Staubli VAL3: Compensated-Y.dtx

public frame fReference = {x=1492.610, y=53.840, z=-416.740, rx=0.091, ry=-0.785, rz=-90.000, fatherId=world[0]}
public jointRx jPark = {j1=0.000, j2=0.000, j3=90.000, j4=0.000, j5=90.000, j6=0.000}
public jointRx jJoint = {j1=3.36880, j2=35.96111, j3=86.31077, j4=-179.94666, j5=-56.93914, j6=-266.65937}
public mdesc mNomSpeed = {accel=100, vel=100, decel=100, tmax=99999, rmax=99999, blend=off, leave=50, reach=50}
public mdesc mSpeed = {tmax=33.3, rmax=100, leave=0.1, reach=0.1, blend=cartesian}
public num nTraj
num nTimeStop
num nTimeStart
num nMode
num nEtat
public pointRx pPoint[1313]
  [0] = {x=-35.000, y=0.000, z=0.000, rx=-0.000, ry=0.000, rz=-0.000, shoulder=lefty, elbow=epositive, wrist=wnegative, fatherId=fReference[0]}
  [1] = {x=-34.500, y=0.000, z=-0.007, rx=-0.000, ry=0.000, rz=-0.000, shoulder=lefty, elbow=epositive, wrist=wnegative, fatherId=fReference[0]}
  [2] = {x=-34.000, y=0.000, z=-0.015, rx=-0.000, ry=0.000, rz=-0.000, shoulder=lefty, elbow=epositive, wrist=wnegative, fatherId=fReference[0]}
  [3] = {x=-33.500, y=0.000, z=-0.022, rx=-0.000, ry=0.000, rz=-0.000, shoulder=lefty, elbow=epositive, wrist=wnegative, fatherId=fReference[0]}
  [4] = {x=-32.999, y=0.000, z=-0.030, rx=-0.000, ry=0.000, rz=-0.000, shoulder=lefty, elbow=epositive, wrist=wnegative, fatherId=fReference[0]}
  [5] = {x=-32.499, y=0.000, z=-0.037, rx=-0.000, ry=0.000, rz=-0.000, shoulder=lefty, elbow=epositive, wrist=wnegative, fatherId=fReference[0]}
  [6] = {x=-31.999, y=0.000, z=-0.045, rx=-0.000, ry=0.000, rz=-0.000, shoulder=lefty, elbow=epositive, wrist=wnegative, fatherId=fReference[0]}
  [7] = {x=-31.499, y=0.000, z=-0.052, rx=-0.000, ry=0.000, rz=-0.000, shoulder=lefty, elbow=epositive, wrist=wnegative, fatherId=fReference[0]}
  [8] = {x=-30.998, y=0.000, z=-0.060, rx=-0.000, ry=0.000, rz=-0.000, shoulder=lefty, elbow=epositive, wrist=wnegative, fatherId=fReference[0]}
  [9] = {x=-30.498, y=0.000, z=-0.067, rx=-0.000, ry=0.000, rz=-0.000, shoulder=lefty, elbow=epositive, wrist=wnegative, fatherId=fReference[0]}
  [10] = {x=-29.998, y=0.000, z=-0.074, rx=-0.000, ry=0.000, rz=-0.000, shoulder=lefty, elbow=epositive, wrist=wnegative, fatherId=fReference[0]}
  [11] = {x=-29.498, y=0.000, z=-0.082, rx=-0.000, ry=0.000, rz=-0.000, shoulder=lefty, elbow=epositive, wrist=wnegative, fatherId=fReference[0]}
  [12] = {x=-28.998, y=0.000, z=-0.089, rx=-0.000, ry=0.000, rz=-0.000, shoulder=lefty, elbow=epositive, wrist=wnegative, fatherId=fReference[0]}
  [13] = {x=-28.498, y=0.000, z=-0.097, rx=-0.000, ry=0.000, rz=-0.000, shoulder=lefty, elbow=epositive, wrist=wnegative, fatherId=fReference[0]}
  [14] = {x=-27.997, y=0.000, z=-0.104, rx=-0.000, ry=0.000, rz=-0.000, shoulder=lefty, elbow=epositive, wrist=wnegative, fatherId=fReference[0]}
  [15] = {x=-27.497, y=0.000, z=-0.112, rx=-0.000, ry=0.000, rz=-0.000, shoulder=lefty, elbow=epositive, wrist=wnegative, fatherId=fReference[0]}
  [16] = {x=-26.997, y=0.000, z=-0.119, rx=-0.000, ry=0.000, rz=-0.000, shoulder=lefty, elbow=epositive, wrist=wnegative, fatherId=fReference[0]}
  [17] = {x=-26.497, y=0.000, z=-0.126, rx=-0.000, ry=0.000, rz=-0.000, shoulder=lefty, elbow=epositive, wrist=wnegative, fatherId=fReference[0]}
  [18] = {x=-25.997, y=0.000, z=-0.134, rx=-0.000, ry=0.000, rz=-0.000, shoulder=lefty, elbow=epositive, wrist=wnegative, fatherId=fReference[0]}
  [19] = {x=-25.497, y=0.000, z=-0.141, rx=-0.000, ry=0.000, rz=-0.000, shoulder=lefty, elbow=epositive, wrist=wnegative, fatherId=fReference[0]}
  [20] = {x=-24.996, y=0.000, z=-0.149, rx=-0.000, ry=0.000, rz=-0.000, shoulder=lefty, elbow=epositive, wrist=wnegative, fatherId=fReference[0]}
  [21] = {x=-24.496, y=0.000, z=-0.156, rx=-0.000, ry=0.000, rz=-0.000, shoulder=lefty, elbow=epositive, wrist=wnegative, fatherId=fReference[0]}
  [22] = {x=-23.996, y=0.000, z=-0.163, rx=-0.000, ry=0.000, rz=-0.000, shoulder=lefty, elbow=epositive, wrist=wnegative, fatherId=fReference[0]}
  [23] = {x=-23.496, y=0.000, z=-0.171, rx=-0.000, ry=0.000, rz=-0.000, shoulder=lefty, elbow=epositive, wrist=wnegative, fatherId=fReference[0]}
  [24] = {x=-22.996, y=0.000, z=-0.178, rx=-0.000, ry=0.000, rz=-0.000, shoulder=lefty, elbow=epositive, wrist=wnegative, fatherId=fReference[0]}
  [25] = {x=-22.496, y=0.000, z=-0.185, rx=-0.000, ry=0.000, rz=-0.000, shoulder=lefty, elbow=epositive, wrist=wnegative, fatherId=fReference[0]}
  [26] = {x=-21.996, y=0.000, z=-0.193, rx=-0.000, ry=0.000, rz=-0.000, shoulder=lefty, elbow=epositive, wrist=wnegative, fatherId=fReference[0]}
  [27] = {x=-21.495, y=0.000, z=-0.200, rx=-0.000, ry=0.000, rz=-0.000, shoulder=lefty, elbow=epositive, wrist=wnegative, fatherId=fReference[0]}
  [28] = {x=-20.995, y=0.000, z=-0.208, rx=-0.000, ry=0.000, rz=-0.000, shoulder=lefty, elbow=epositive, wrist=wnegative, fatherId=fReference[0]}
  [29] = {x=-20.495, y=0.000, z=-0.215, rx=-0.000, ry=0.000, rz=-0.000, shoulder=lefty, elbow=epositive, wrist=wnegative, fatherId=fReference[0]}
  [30] = {x=-19.995, y=0.000, z=-0.222, rx=-0.000, ry=0.000, rz=-0.000, shoulder=lefty, elbow=epositive, wrist=wnegative, fatherId=fReference[0]}
  [31] = {x=-19.495, y=0.000, z=-0.230, rx=-0.000, ry=0.000, rz=-0.000, shoulder=lefty, elbow=epositive, wrist=wnegative, fatherId=fReference[0]}
  [32] = {x=-18.995, y=0.000, z=-0.237, rx=-0.000, ry=0.000, rz=-0.000, shoulder=lefty, elbow=epositive, wrist=wnegative, fatherId=fReference[0]}
  [33] = {x=-18.495, y=0.000, z=-0.244, rx=-0.000, ry=0.000, rz=-0.000, shoulder=lefty, elbow=epositive, wrist=wnegative, fatherId=fReference[0]}
  [34] = {x=-17.995, y=0.000, z=-0.252, rx=-0.000, ry=0.000, rz=-0.000, shoulder=lefty, elbow=epositive, wrist=wnegative, fatherId=fReference[0]}
  [35] = {x=-17.494, y=0.000, z=-0.259, rx=-0.000, ry=0.000, rz=-0.000, shoulder=lefty, elbow=epositive, wrist=wnegative, fatherId=fReference[0]}
  [36] = {x=-16.994, y=0.000, z=-0.266, rx=-0.000, ry=0.000, rz=-0.000, shoulder=lefty, elbow=epositive, wrist=wnegative, fatherId=fReference[0]}
  [37] = {x=-16.494, y=0.000, z=-0.274, rx=-0.000, ry=0.000, rz=-0.000, shoulder=lefty, elbow=epositive, wrist=wnegative, fatherId=fReference[0]}
  [38] = {x=-15.994, y=0.000, z=-0.281, rx=-0.000, ry=0.000, rz=-0.000, shoulder=lefty, elbow=epositive, wrist=wnegative, fatherId=fReference[0]}
  [39] = {x=-15.494, y=0.000, z=-0.288, rx=-0.000, ry=0.000, rz=-0.000, shoulder=lefty, elbow=epositive, wrist=wnegative, fatherId=fReference[0]}
  [40] = {x=-14.994, y=0.000, z=-0.296, rx=-0.000, ry=0.000, rz=-0.000, shoulder=lefty, elbow=epositive, wrist=wnegative, fatherId=fReference[0]}
  [41] = {x=-14.494, y=0.000, z=-0.303, rx=-0.000, ry=0.000, rz=-0.000, shoulder=lefty, elbow=epositive, wrist=wnegative, fatherId=fReference[0]}
  [42] = {x=-13.994, y=0.000, z=-0.310, rx=-0.000, ry=0.000, rz=-0.000, shoulder=lefty, elbow=epositive, wrist=wnegative, fatherId=fReference[0]}
  [43] = {x=-13.493, y=0.000, z=-0.318, rx=-0.000, ry=0.000, rz=-0.000, shoulder=lefty, elbow=epositive, wrist=wnegative, fatherId=fReference[0]}
  [44] = {x=-12.993, y=0.000, z=-0.325, rx=-0.000, ry=0.000, rz=-0.000, shoulder=lefty, elbow=epositive, wrist=wnegative, fatherId=fReference[0]}
  [45] = {x=-12.493, y=0.000, z=-0.332, rx=-0.000, ry=0.000, rz=-0.000, shoulder=lefty, elbow=epositive, wrist=wnegative, fatherId=fReference[0]}
  [46] = {x=-11.993, y=0.000, z=-0.340, rx=-0.000, ry=0.000, rz=-0.000, shoulder=lefty, elbow=epositive, wrist=wnegative, fatherId=fReference[0]}
  [47] = {x=-11.493, y=0.000, z=-0.347, rx=-0.000, ry=0.000, rz=-0.000, shoulder=lefty, elbow=epositive, wrist=wnegative, fatherId=fReference[0]}
  [48] = {x=-10.993, y=0.000, z=-0.354, rx=-0.000, ry=0.000, rz=-0.000, shoulder=lefty, elbow=epositive, wrist=wnegative, fatherId=fReference[0]}
  [49] = {x=-10.493, y=0.000, z=-0.362, rx=-0.000, ry=0.000, rz=-0.000, shoulder=lefty, elbow=epositive, wrist=wnegative, fatherId=fReference[0]}
  [50] = {x=-9.993, y=0.000, z=-0.369, rx=-0.000, ry=0.000, rz=-0.000, shoulder=lefty, elbow=epositive, wrist=wnegative, fatherId=fReference[0]}
  [51] = {x=-9.492, y=0.000, z=-0.377, rx=-0.000, ry=0.000, rz=-0.000, shoulder=lefty, elbow=epositive, wrist=wnegative, fatherId=fReference[0]}
  [52] = {x=-8.992, y=0.000, z=-0.384, rx=-0.000, ry=0.000, rz=-0.000, shoulder=lefty, elbow=epositive, wrist=wnegative, fatherId=fReference[0]}
  [53] = {x=-8.492, y=0.000, z=-0.391, rx=-0.000, ry=0.000, rz=-0.000, shoulder=lefty, elbow=epositive, wrist=wnegative, fatherId=fReference[0]}
  [54] = {x=-7.992, y=0.000, z=-0.399, rx=-0.000, ry=0.000, rz=-0.000, shoulder=lefty, elbow=epositive, wrist=wnegative, fatherId=fReference[0]}
  [55] = {x=-7.492, y=0.000, z=-0.406, rx=-0.000, ry=0.000, rz=-0.000, shoulder=lefty, elbow=epositive, wrist=wnegative, fatherId=fReference[0]}
  [56] = {x=-6.992, y=0.000, z=-0.413, rx=-0.000, ry=0.000, rz=-0.000, shoulder=lefty, elbow=epositive, wrist=wnegative, fatherId=fReference[0]}
  [57] = {x=-6.492, y=0.000, z=-0.421, rx=-0.000, ry=0.000, rz=-0.000, shoulder=lefty, elbow=epositive, wrist=wnegative, fatherId=fReference[0]}
  [58] = {x=-5.991, y=0.000, z=-0.428, rx=-0.000, ry=0.000, rz=-0.000, shoulder=lefty, elbow=epositive, wrist=wnegative, fatherId=fReference[0]}
  [59] = {x=-5.491, y=0.000, z=-0.435, rx=-0.000, ry=0.000, rz=-0.000, shoulder=lefty, elbow=epositive, wrist=wnegative, fatherId=fReference[0]}
  [60] = {x=-4.991, y=0.000, z=-0.443, rx=-0.000, ry=0.000, rz=-0.000, shoulder=lefty, elbow=epositive, wrist=wnegative, fatherId=fReference[0]}
  [61] = {x=-4.491, y=0.000, z=-0.450, rx=-0.000, ry=0.000, rz=-0.000, shoulder=lefty, elbow=epositive, wrist=wnegative, fatherId=fReference[0]}
  [62] = {x=-3.991, y=0.000, z=-0.458, rx=-0.000, ry=0.000, rz=-0.000, shoulder=lefty, elbow=epositive, wrist=wnegative, fatherId=fReference[0]}
  [63] = {x=-3.491, y=0.000, z=-0.465, rx=-0.000, ry=0.000, rz=-0.000, shoulder=lefty, elbow=epositive, wrist=wnegative, fatherId=fReference[0]}
  [64] = {x=-2.991, y=0.000, z=-0.472, rx=-0.000, ry=0.000, rz=-0.000, shoulder=lefty, elbow=epositive, wrist=wnegative, fatherId=fReference[0]}
  [65] = {x=-2.490, y=0.000, z=-0.480, rx=-0.000, ry=0.000, rz=-0.000, shoulder=lefty, elbow=epositive, wrist=wnegative, fatherId=fReference[0]}
  [66] = {x=-1.990, y=0.000, z=-0.487, rx=-0.000, ry=0.000, rz=-0.000, shoulder=lefty, elbow=epositive, wrist=wnegative, fatherId=fReference[0]}
  [67] = {x=-1.490, y=0.000, z=-0.495, rx=-0.000, ry=0.000, rz=-0.000, shoulder=lefty, elbow=epositive, wrist=wnegative, fatherId=fReference[0]}
  [68] = {x=-0.990, y=0.000, z=-0.502, rx=-0.000, ry=0.000, rz=-0.000, shoulder=lefty, elbow=epositive, wrist=wnegative, fatherId=fReference[0]}
  [69] = {x=-0.490, y=0.000, z=-0.509, rx=-0.000, ry=0.000, rz=-0.000, shoulder=lefty, elbow=epositive, wrist=wnegative, fatherId=fReference[0]}
  [70] = {x=0.010, y=0.000, z=-0.517, rx=-0.000, ry=0.000, rz=-0.000, shoulder=lefty, elbow=epositive, wrist=wnegative, fatherId=fReference[0]}
  [71] = {x=0.511, y=0.000, z=-0.524, rx=-0.000, ry=0.000, rz=-0.000, shoulder=lefty, elbow=epositive, wrist=wnegative, fatherId=fReference[0]}
  [72] = {x=1.011, y=0.000, z=-0.532, rx=-0.000, ry=0.000, rz=-0.000, shoulder=lefty, elbow=epositive, wrist=wnegative, fatherId=fReference[0]}
  [73] = {x=1.511, y=0.000, z=-0.539, rx=-0.000, ry=0.000, rz=-0.000, shoulder=lefty, elbow=epositive, wrist=wnegative, fatherId=fReference[0]}
  [74] = {x=2.011, y=0.000, z=-0.547, rx=-0.000, ry=0.000, rz=-0.000, shoulder=lefty, elbow=epositive, wrist=wnegative, fatherId=fReference[0]}
  [75] = {x=2.511, y=0.000, z=-0.554, rx=-0.000, ry=0.000, rz=-0.000, shoulder=lefty, elbow=epositive, wrist=wnegative, fatherId=fReference[0]}
  [76] = {x=3.012, y=0.000, z=-0.562, rx=-0.000, ry=0.000, rz=-0.000, shoulder=lefty, elbow=epositive, wrist=wnegative, fatherId=fReference[0]}
  [77] = {x=3.512, y=0.000, z=-0.569, rx=-0.000, ry=0.000, rz=-0.000, shoulder=lefty, elbow=epositive, wrist=wnegative, fatherId=fReference[0]}
  [78] = {x=4.012, y=0.000, z=-0.576, rx=-0.000, ry=0.000, rz=-0.000, shoulder=lefty, elbow=epositive, wrist=wnegative, fatherId=fReference[0]}
  [79] = {x=4.512, y=0.000, z=-0.584, rx=-0.000, ry=0.000, rz=-0.000, shoulder=lefty, elbow=epositive, wrist=wnegative, fatherId=fReference[0]}
  [80] = {x=5.012, y=0.000, z=-0.591, rx=-0.000, ry=0.000, rz=-0.000, shoulder=lefty, elbow=epositive, wrist=wnegative, fatherId=fReference[0]}
  [81] = {x=5.513, y=0.000, z=-0.599, rx=-0.000, ry=0.000, rz=-0.000, shoulder=lefty, elbow=epositive, wrist=wnegative, fatherId=fReference[0]}
  [82] = {x=6.013, y=0.000, z=-0.606, rx=-0.000, ry=0.000, rz=-0.000, shoulder=lefty, elbow=epositive, wrist=wnegative, fatherId=fReference[0]}
  [83] = {x=6.513, y=0.000, z=-0.614, rx=-0.000, ry=0.000, rz=-0.000, shoulder=lefty, elbow=epositive, wrist=wnegative, fatherId=fReference[0]}
  [84] = {x=7.013, y=0.000, z=-0.621, rx=-0.000, ry=0.000, rz=-0.000, shoulder=lefty, elbow=epositive, wrist=wnegative, fatherId=fReference[0]}
  [85] = {x=7.514, y=0.000, z=-0.629, rx=-0.000, ry=0.000, rz=-0.000, shoulder=lefty, elbow=epositive, wrist=wnegative, fatherId=fReference[0]}
  [86] = {x=8.014, y=0.000, z=-0.637, rx=-0.000, ry=0.000, rz=-0.000, shoulder=lefty, elbow=epositive, wrist=wnegative, fatherId=fReference[0]}
  [87] = {x=8.514, y=0.000, z=-0.644, rx=-0.000, ry=0.000, rz=-0.000, shoulder=lefty, elbow=epositive, wrist=wnegative, fatherId=fReference[0]}
  [88] = {x=9.014, y=0.000, z=-0.652, rx=-0.000, ry=0.000, rz=-0.000, shoulder=lefty, elbow=epositive, wrist=wnegative, fatherId=fReference[0]}
  [89] = {x=9.515, y=0.000, z=-0.659, rx=-0.000, ry=0.000, rz=-0.000, shoulder=lefty, elbow=epositive, wrist=wnegative, fatherId=fReference[0]}
  [90] = {x=10.015, y=0.000, z=-0.667, rx=-0.000, ry=0.000, rz=-0.000, shoulder=lefty, elbow=epositive, wrist=wnegative, fatherId=fReference[0]}
  [91] = {x=10.515, y=0.000, z=-0.674, rx=-0.000, ry=0.000, rz=-0.000, shoulder=lefty, elbow=epositive, wrist=wnegative, fatherId=fReference[0]}
  [92] = {x=11.016, y=0.000, z=-0.682, rx=-0.000, ry=0.000, rz=-0.000, shoulder=lefty, elbow=epositive, wrist=wnegative, fatherId=fReference[0]}
  [93] = {x=11.516, y=0.000, z=-0.690, rx=-0.000, ry=0.000, rz=-0.000, shoulder=lefty, elbow=epositive, wrist=wnegative, fatherId=fReference[0]}
  [94] = {x=12.016, y=0.000, z=-0.697, rx=-0.000, ry=0.000, rz=-0.000, shoulder=lefty, elbow=epositive, wrist=wnegative, fatherId=fReference[0]}
  [95] = {x=12.516, y=0.000, z=-0.705, rx=-0.000, ry=0.000, rz=-0.000, shoulder=lefty, elbow=epositive, wrist=wnegative, fatherId=fReference[0]}
  [96] = {x=13.017, y=0.000, z=-0.713, rx=-0.000, ry=0.000, rz=-0.000, shoulder=lefty, elbow=epositive, wrist=wnegative, fatherId=fReference[0]}
  [97] = {x=13.517, y=0.000, z=-0.720, rx=-0.000, ry=0.000, rz=-0.000, shoulder=lefty, elbow=epositive, wrist=wnegative, fatherId=fReference[0]}
  [98] = {x=14.017, y=0.000, z=-0.728, rx=-0.000, ry=0.000, rz=-0.000, shoulder=lefty, elbow=epositive, wrist=wnegative, fatherId=fReference[0]}
  [99] = {x=14.518, y=0.000, z=-0.736, rx=-0.000, ry=0.000, rz=-0.000, shoulder=lefty, elbow=epositive, wrist=wnegative, fatherId=fReference[0]}
  [100] = {x=15.018, y=0.000, z=-0.743, rx=-0.000, ry=0.000, rz=-0.000, shoulder=lefty, elbow=epositive, wrist=wnegative, fatherId=fReference[0]}
  [101] = {x=15.519, y=0.000, z=-0.751, rx=-0.000, ry=0.000, rz=-0.000, shoulder=lefty, elbow=epositive, wrist=wnegative, fatherId=fReference[0]}
  [102] = {x=16.019, y=0.000, z=-0.759, rx=-0.000, ry=0.000, rz=-0.000, shoulder=lefty, elbow=epositive, wrist=wnegative, fatherId=fReference[0]}
  [103] = {x=16.519, y=0.000, z=-0.766, rx=-0.000, ry=0.000, rz=-0.000, shoulder=lefty, elbow=epositive, wrist=wnegative, fatherId=fReference[0]}
  [104] = {x=17.020, y=0.000, z=-0.774, rx=-0.000, ry=0.000, rz=-0.000, shoulder=lefty, elbow=epositive, wrist=wnegative, fatherId=fReference[0]}
  [105] = {x=17.520, y=0.000, z=-0.782, rx=-0.000, ry=0.000, rz=-0.000, shoulder=lefty, elbow=epositive, wrist=wnegative, fatherId=fReference[0]}
  [106] = {x=18.020, y=0.000, z=-0.790, rx=-0.000, ry=0.000, rz=-0.000, shoulder=lefty, elbow=epositive, wrist=wnegative, fatherId=fReference[0]}
  [107] = {x=18.521, y=0.000, z=-0.798, rx=-0.000, ry=0.000, rz=-0.000, shoulder=lefty, elbow=epositive, wrist=wnegative, fatherId=fReference[0]}
  [108] = {x=19.021, y=0.000, z=-0.805, rx=-0.000, ry=0.000, rz=-0.000, shoulder=lefty, elbow=epositive, wrist=wnegative, fatherId=fReference[0]}
  [109] = {x=19.522, y=0.000, z=-0.813, rx=-0.000, ry=0.000, rz=-0.000, shoulder=lefty, elbow=epositive, wrist=wnegative, fatherId=fReference[0]}
  [110] = {x=20.022, y=0.000, z=-0.821, rx=-0.000, ry=0.000, rz=-0.000, shoulder=lefty, elbow=epositive, wrist=wnegative, fatherId=fReference[0]}
  [111] = {x=20.523, y=0.000, z=-0.829, rx=-0.000, ry=0.000, rz=-0.000, shoulder=lefty, elbow=epositive, wrist=wnegative, fatherId=fReference[0]}
  [112] = {x=21.023, y=0.000, z=-0.837, rx=-0.000, ry=0.000, rz=-0.000, shoulder=lefty, elbow=epositive, wrist=wnegative, fatherId=fReference[0]}
  [113] = {x=21.524, y=0.000, z=-0.845, rx=-0.000, ry=0.000, rz=-0.000, shoulder=lefty, elbow=epositive, wrist=wnegative, fatherId=fReference[0]}
  [114] = {x=22.024, y=0.000, z=-0.853, rx=-0.000, ry=0.000, rz=-0.000, shoulder=lefty, elbow=epositive, wrist=wnegative, fatherId=fReference[0]}
  [115] = {x=22.525, y=0.000, z=-0.861, rx=-0.000, ry=0.000, rz=-0.000, shoulder=lefty, elbow=epositive, wrist=wnegative, fatherId=fReference[0]}
  [116] = {x=23.025, y=0.000, z=-0.869, rx=-0.000, ry=0.000, rz=-0.000, shoulder=lefty, elbow=epositive, wrist=wnegative, fatherId=fReference[0]}
  [117] = {x=23.526, y=0.000, z=-0.877, rx=-0.000, ry=0.000, rz=-0.000, shoulder=lefty, elbow=epositive, wrist=wnegative, fatherId=fReference[0]}
  [118] = {x=24.026, y=0.000, z=-0.885, rx=-0.000, ry=0.000, rz=-0.000, shoulder=lefty, elbow=epositive, wrist=wnegative, fatherId=fReference[0]}
  [119] = {x=24.527, y=0.000, z=-0.893, rx=-0.000, ry=0.000, rz=-0.000, shoulder=lefty, elbow=epositive, wrist=wnegative, fatherId=fReference[0]}
  [120] = {x=25.028, y=0.000, z=-0.901, rx=-0.000, ry=0.000, rz=-0.000, shoulder=lefty, elbow=epositive, wrist=wnegative, fatherId=fReference[0]}
  [121] = {x=25.528, y=0.000, z=-0.909, rx=-0.000, ry=0.000, rz=-0.000, shoulder=lefty, elbow=epositive, wrist=wnegative, fatherId=fReference[0]}
  [122] = {x=26.029, y=0.000, z=-0.917, rx=-0.000, ry=0.000, rz=-0.000, shoulder=lefty, elbow=epositive, wrist=wnegative, fatherId=fReference[0]}
  [123] = {x=26.530, y=0.000, z=-0.925, rx=-0.000, ry=0.000, rz=-0.000, shoulder=lefty, elbow=epositive, wrist=wnegative, fatherId=fReference[0]}
  [124] = {x=27.030, y=0.000, z=-0.933, rx=-0.000, ry=0.000, rz=-0.000, shoulder=lefty, elbow=epositive, wrist=wnegative, fatherId=fReference[0]}
  [125] = {x=27.531, y=0.000, z=-0.941, rx=-0.000, ry=0.000, rz=-0.000, shoulder=lefty, elbow=epositive, wrist=wnegative, fatherId=fReference[0]}
  [126] = {x=28.032, y=0.000, z=-0.950, rx=-0.000, ry=0.000, rz=-0.000, shoulder=lefty, elbow=epositive, wrist=wnegative, fatherId=fReference[0]}
  [127] = {x=28.532, y=0.000, z=-0.958, rx=-0.000, ry=0.000, rz=-0.000, shoulder=lefty, elbow=epositive, wrist=wnegative, fatherId=fReference[0]}
  [128] = {x=29.033, y=0.000, z=-0.966, rx=-0.000, ry=0.000, rz=-0.000, shoulder=lefty, elbow=epositive, wrist=wnegative, fatherId=fReference[0]}
  [129] = {x=29.534, y=0.000, z=-0.974, rx=-0.000, ry=0.000, rz=-0.000, shoulder=lefty, elbow=epositive, wrist=wnegative, fatherId=fReference[0]}
  [130] = {x=30.035, y=0.000, z=-0.983, rx=-0.000, ry=0.000, rz=-0.000, shoulder=lefty, elbow=epositive, wrist=wnegative, fatherId=fReference[0]}
  [131] = {x=30.536, y=0.000, z=-0.991, rx=-0.000, ry=0.000, rz=-0.000, shoulder=lefty, elbow=epositive, wrist=wnegative, fatherId=fReference[0]}
  [132] = {x=31.036, y=0.000, z=-1.000, rx=-0.000, ry=0.000, rz=-0.000, shoulder=lefty, elbow=epositive, wrist=wnegative, fatherId=fReference[0]}
  [133] = {x=31.537, y=0.000, z=-1.008, rx=-0.000, ry=0.000, rz=-0.000, shoulder=lefty, elbow=epositive, wrist=wnegative, fatherId=fReference[0]}
  [134] = {x=32.038, y=0.000, z=-1.016, rx=-0.000, ry=0.000, rz=-0.000, shoulder=lefty, elbow=epositive, wrist=wnegative, fatherId=fReference[0]}
  [135] = {x=32.539, y=0.000, z=-1.025, rx=-0.000, ry=0.000, rz=-0.000, shoulder=lefty, elbow=epositive, wrist=wnegative, fatherId=fReference[0]}
  [136] = {x=33.040, y=0.000, z=-1.034, rx=-0.000, ry=0.000, rz=-0.000, shoulder=lefty, elbow=epositive, wrist=wnegative, fatherId=fReference[0]}
  [137] = {x=33.541, y=0.000, z=-1.042, rx=-0.000, ry=0.000, rz=-0.000, shoulder=lefty, elbow=epositive, wrist=wnegative, fatherId=fReference[0]}
  [138] = {x=34.042, y=0.000, z=-1.051, rx=-0.000, ry=0.000, rz=-0.000, shoulder=lefty, elbow=epositive, wrist=wnegative, fatherId=fReference[0]}
  [139] = {x=34.543, y=0.000, z=-1.060, rx=-0.000, ry=0.000, rz=-0.000, shoulder=lefty, elbow=epositive, wrist=wnegative, fatherId=fReference[0]}
  [140] = {x=35.026, y=0.000, z=-1.067, rx=-0.000, ry=0.000, rz=-0.000, shoulder=lefty, elbow=epositive, wrist=wnegative, fatherId=fReference[0]}
  [141] = {x=34.526, y=0.000, z=-1.073, rx=-0.000, ry=0.000, rz=-0.000, shoulder=lefty, elbow=epositive, wrist=wnegative, fatherId=fReference[0]}
  [142] = {x=34.026, y=0.000, z=-1.080, rx=-0.000, ry=0.000, rz=-0.000, shoulder=lefty, elbow=epositive, wrist=wnegative, fatherId=fReference[0]}
  [143] = {x=33.525, y=0.000, z=-1.086, rx=-0.000, ry=0.000, rz=-0.000, shoulder=lefty, elbow=epositive, wrist=wnegative, fatherId=fReference[0]}
  [144] = {x=33.025, y=0.000, z=-1.093, rx=-0.000, ry=0.000, rz=-0.000, shoulder=lefty, elbow=epositive, wrist=wnegative, fatherId=fReference[0]}
  [145] = {x=32.525, y=0.000, z=-1.100, rx=-0.000, ry=0.000, rz=-0.000, shoulder=lefty, elbow=epositive, wrist=wnegative, fatherId=fReference[0]}
  [146] = {x=32.025, y=0.000, z=-1.107, rx=-0.000, ry=0.000, rz=-0.000, shoulder=lefty, elbow=epositive, wrist=wnegative, fatherId=fReference[0]}
  [147] = {x=31.524, y=0.000, z=-1.114, rx=-0.000, ry=0.000, rz=-0.000, shoulder=lefty, elbow=epositive, wrist=wnegative, fatherId=fReference[0]}
  [148] = {x=31.024, y=0.000, z=-1.121, rx=-0.000, ry=0.000, rz=-0.000, shoulder=lefty, elbow=epositive, wrist=wnegative, fatherId=fReference[0]}
  [149] = {x=30.524, y=0.000, z=-1.127, rx=-0.000, ry=0.000, rz=-0.000, shoulder=lefty, elbow=epositive, wrist=wnegative, fatherId=fReference[0]}
  [150] = {x=30.024, y=0.000, z=-1.135, rx=-0.000, ry=0.000, rz=-0.000, shoulder=lefty, elbow=epositive, wrist=wnegative, fatherId=fReference[0]}
  [151] = {x=29.524, y=0.000, z=-1.141, rx=-0.000, ry=0.000, rz=-0.000, shoulder=lefty, elbow=epositive, wrist=wnegative, fatherId=fReference[0]}
  [152] = {x=29.024, y=0.000, z=-1.149, rx=-0.000, ry=0.000, rz=-0.000, shoulder=lefty, elbow=epositive, wrist=wnegative, fatherId=fReference[0]}
  [153] = {x=28.523, y=0.000, z=-1.155, rx=-0.000, ry=0.000, rz=-0.000, shoulder=lefty, elbow=epositive, wrist=wnegative, fatherId=fReference[0]}
  [154] = {x=28.023, y=0.000, z=-1.163, rx=-0.000, ry=0.000, rz=-0.000, shoulder=lefty, elbow=epositive, wrist=wnegative, fatherId=fReference[0]}
  [155] = {x=27.523, y=0.000, z=-1.170, rx=-0.000, ry=0.000, rz=-0.000, shoulder=lefty, elbow=epositive, wrist=wnegative, fatherId=fReference[0]}
  [156] = {x=27.023, y=0.000, z=-1.177, rx=-0.000, ry=0.000, rz=-0.000, shoulder=lefty, elbow=epositive, wrist=wnegative, fatherId=fReference[0]}
  [157] = {x=26.523, y=0.000, z=-1.184, rx=-0.000, ry=0.000, rz=-0.000, shoulder=lefty, elbow=epositive, wrist=wnegative, fatherId=fReference[0]}
  [158] = {x=26.023, y=0.000, z=-1.191, rx=-0.000, ry=0.000, rz=-0.000, shoulder=lefty, elbow=epositive, wrist=wnegative, fatherId=fReference[0]}
  [159] = {x=25.523, y=0.000, z=-1.198, rx=-0.000, ry=0.000, rz=-0.000, shoulder=lefty, elbow=epositive, wrist=wnegative, fatherId=fReference[0]}
  [160] = {x=25.023, y=0.000, z=-1.205, rx=-0.000, ry=0.000, rz=-0.000, shoulder=lefty, elbow=epositive, wrist=wnegative, fatherId=fReference[0]}
  [161] = {x=24.523, y=0.000, z=-1.212, rx=-0.000, ry=0.000, rz=-0.000, shoulder=lefty, elbow=epositive, wrist=wnegative, fatherId=fReference[0]}
  [162] = {x=24.023, y=0.000, z=-1.219, rx=-0.000, ry=0.000, rz=-0.000, shoulder=lefty, elbow=epositive, wrist=wnegative, fatherId=fReference[0]}
  [163] = {x=23.523, y=0.000, z=-1.227, rx=-0.000, ry=0.000, rz=-0.000, shoulder=lefty, elbow=epositive, wrist=wnegative, fatherId=fReference[0]}
  [164] = {x=23.023, y=0.000, z=-1.234, rx=-0.000, ry=0.000, rz=-0.000, shoulder=lefty, elbow=epositive, wrist=wnegative, fatherId=fReference[0]}
  [165] = {x=22.523, y=0.000, z=-1.241, rx=-0.000, ry=0.000, rz=-0.000, shoulder=lefty, elbow=epositive, wrist=wnegative, fatherId=fReference[0]}
  [166] = {x=22.022, y=0.000, z=-1.248, rx=-0.000, ry=0.000, rz=-0.000, shoulder=lefty, elbow=epositive, wrist=wnegative, fatherId=fReference[0]}
  [167] = {x=21.522, y=0.000, z=-1.255, rx=-0.000, ry=0.000, rz=-0.000, shoulder=lefty, elbow=epositive, wrist=wnegative, fatherId=fReference[0]}
  [168] = {x=21.022, y=0.000, z=-1.262, rx=-0.000, ry=0.000, rz=-0.000, shoulder=lefty, elbow=epositive, wrist=wnegative, fatherId=fReference[0]}
  [169] = {x=20.522, y=0.000, z=-1.270, rx=-0.000, ry=0.000, rz=-0.000, shoulder=lefty, elbow=epositive, wrist=wnegative, fatherId=fReference[0]}
  [170] = {x=20.022, y=0.000, z=-1.277, rx=-0.000, ry=0.000, rz=-0.000, shoulder=lefty, elbow=epositive, wrist=wnegative, fatherId=fReference[0]}
  [171] = {x=19.522, y=0.000, z=-1.284, rx=-0.000, ry=0.000, rz=-0.000, shoulder=lefty, elbow=epositive, wrist=wnegative, fatherId=fReference[0]}
  [172] = {x=19.022, y=0.000, z=-1.292, rx=-0.000, ry=0.000, rz=-0.000, shoulder=lefty, elbow=epositive, wrist=wnegative, fatherId=fReference[0]}
  [173] = {x=18.522, y=0.000, z=-1.299, rx=-0.000, ry=0.000, rz=-0.000, shoulder=lefty, elbow=epositive, wrist=wnegative, fatherId=fReference[0]}
  [174] = {x=18.022, y=0.000, z=-1.306, rx=-0.000, ry=0.000, rz=-0.000, shoulder=lefty, elbow=epositive, wrist=wnegative, fatherId=fReference[0]}
  [175] = {x=17.522, y=0.000, z=-1.313, rx=-0.000, ry=0.000, rz=-0.000, shoulder=lefty, elbow=epositive, wrist=wnegative, fatherId=fReference[0]}
  [176] = {x=17.022, y=0.000, z=-1.321, rx=-0.000, ry=0.000, rz=-0.000, shoulder=lefty, elbow=epositive, wrist=wnegative, fatherId=fReference[0]}
  [177] = {x=16.522, y=0.000, z=-1.328, rx=-0.000, ry=0.000, rz=-0.000, shoulder=lefty, elbow=epositive, wrist=wnegative, fatherId=fReference[0]}
  [178] = {x=16.022, y=0.000, z=-1.335, rx=-0.000, ry=0.000, rz=-0.000, shoulder=lefty, elbow=epositive, wrist=wnegative, fatherId=fReference[0]}
  [179] = {x=15.522, y=0.000, z=-1.343, rx=-0.000, ry=0.000, rz=-0.000, shoulder=lefty, elbow=epositive, wrist=wnegative, fatherId=fReference[0]}
  [180] = {x=15.022, y=0.000, z=-1.350, rx=-0.000, ry=0.000, rz=-0.000, shoulder=lefty, elbow=epositive, wrist=wnegative, fatherId=fReference[0]}
  [181] = {x=14.522, y=0.000, z=-1.357, rx=-0.000, ry=0.000, rz=-0.000, shoulder=lefty, elbow=epositive, wrist=wnegative, fatherId=fReference[0]}
  [182] = {x=14.022, y=0.000, z=-1.365, rx=-0.000, ry=0.000, rz=-0.000, shoulder=lefty, elbow=epositive, wrist=wnegative, fatherId=fReference[0]}
  [183] = {x=13.523, y=0.000, z=-1.372, rx=-0.000, ry=0.000, rz=-0.000, shoulder=lefty, elbow=epositive, wrist=wnegative, fatherId=fReference[0]}
  [184] = {x=13.023, y=0.000, z=-1.380, rx=-0.000, ry=0.000, rz=-0.000, shoulder=lefty, elbow=epositive, wrist=wnegative, fatherId=fReference[0]}
  [185] = {x=12.523, y=0.000, z=-1.387, rx=-0.000, ry=0.000, rz=-0.000, shoulder=lefty, elbow=epositive, wrist=wnegative, fatherId=fReference[0]}
  [186] = {x=12.023, y=0.000, z=-1.395, rx=-0.000, ry=0.000, rz=-0.000, shoulder=lefty, elbow=epositive, wrist=wnegative, fatherId=fReference[0]}
  [187] = {x=11.523, y=0.000, z=-1.402, rx=-0.000, ry=0.000, rz=-0.000, shoulder=lefty, elbow=epositive, wrist=wnegative, fatherId=fReference[0]}
  [188] = {x=11.023, y=0.000, z=-1.409, rx=-0.000, ry=0.000, rz=-0.000, shoulder=lefty, elbow=epositive, wrist=wnegative, fatherId=fReference[0]}
  [189] = {x=10.523, y=0.000, z=-1.417, rx=-0.000, ry=0.000, rz=-0.000, shoulder=lefty, elbow=epositive, wrist=wnegative, fatherId=fReference[0]}
  [190] = {x=10.023, y=0.000, z=-1.424, rx=-0.000, ry=0.000, rz=-0.000, shoulder=lefty, elbow=epositive, wrist=wnegative, fatherId=fReference[0]}
  [191] = {x=9.523, y=0.000, z=-1.432, rx=-0.000, ry=0.000, rz=-0.000, shoulder=lefty, elbow=epositive, wrist=wnegative, fatherId=fReference[0]}
  [192] = {x=9.023, y=0.000, z=-1.439, rx=-0.000, ry=0.000, rz=-0.000, shoulder=lefty, elbow=epositive, wrist=wnegative, fatherId=fReference[0]}
  [193] = {x=8.523, y=0.000, z=-1.447, rx=-0.000, ry=0.000, rz=-0.000, shoulder=lefty, elbow=epositive, wrist=wnegative, fatherId=fReference[0]}
  [194] = {x=8.023, y=0.000, z=-1.454, rx=-0.000, ry=0.000, rz=-0.000, shoulder=lefty, elbow=epositive, wrist=wnegative, fatherId=fReference[0]}
  [195] = {x=7.523, y=0.000, z=-1.462, rx=-0.000, ry=0.000, rz=-0.000, shoulder=lefty, elbow=epositive, wrist=wnegative, fatherId=fReference[0]}
  [196] = {x=7.023, y=0.000, z=-1.469, rx=-0.000, ry=0.000, rz=-0.000, shoulder=lefty, elbow=epositive, wrist=wnegative, fatherId=fReference[0]}
  [197] = {x=6.523, y=0.000, z=-1.477, rx=-0.000, ry=0.000, rz=-0.000, shoulder=lefty, elbow=epositive, wrist=wnegative, fatherId=fReference[0]}
  [198] = {x=6.023, y=0.000, z=-1.484, rx=-0.000, ry=0.000, rz=-0.000, shoulder=lefty, elbow=epositive, wrist=wnegative, fatherId=fReference[0]}
  [199] = {x=5.524, y=0.000, z=-1.492, rx=-0.000, ry=0.000, rz=-0.000, shoulder=lefty, elbow=epositive, wrist=wnegative, fatherId=fReference[0]}
  [200] = {x=5.024, y=0.000, z=-1.500, rx=-0.000, ry=0.000, rz=-0.000, shoulder=lefty, elbow=epositive, wrist=wnegative, fatherId=fReference[0]}
  [201] = {x=4.524, y=0.000, z=-1.507, rx=-0.000, ry=0.000, rz=-0.000, shoulder=lefty, elbow=epositive, wrist=wnegative, fatherId=fReference[0]}
  [202] = {x=4.024, y=0.000, z=-1.515, rx=-0.000, ry=0.000, rz=-0.000, shoulder=lefty, elbow=epositive, wrist=wnegative, fatherId=fReference[0]}
  [203] = {x=3.524, y=0.000, z=-1.522, rx=-0.000, ry=0.000, rz=-0.000, shoulder=lefty, elbow=epositive, wrist=wnegative, fatherId=fReference[0]}
  [204] = {x=3.024, y=0.000, z=-1.530, rx=-0.000, ry=0.000, rz=-0.000, shoulder=lefty, elbow=epositive, wrist=wnegative, fatherId=fReference[0]}
  [205] = {x=2.524, y=0.000, z=-1.538, rx=-0.000, ry=0.000, rz=-0.000, shoulder=lefty, elbow=epositive, wrist=wnegative, fatherId=fReference[0]}
  [206] = {x=2.024, y=0.000, z=-1.545, rx=-0.000, ry=0.000, rz=-0.000, shoulder=lefty, elbow=epositive, wrist=wnegative, fatherId=fReference[0]}
  [207] = {x=1.524, y=0.000, z=-1.553, rx=-0.000, ry=0.000, rz=-0.000, shoulder=lefty, elbow=epositive, wrist=wnegative, fatherId=fReference[0]}
  [208] = {x=1.024, y=0.000, z=-1.561, rx=-0.000, ry=0.000, rz=-0.000, shoulder=lefty, elbow=epositive, wrist=wnegative, fatherId=fReference[0]}
  [209] = {x=0.525, y=0.000, z=-1.568, rx=-0.000, ry=0.000, rz=-0.000, shoulder=lefty, elbow=epositive, wrist=wnegative, fatherId=fReference[0]}
  [210] = {x=0.025, y=0.000, z=-1.576, rx=-0.000, ry=0.000, rz=-0.000, shoulder=lefty, elbow=epositive, wrist=wnegative, fatherId=fReference[0]}
  [211] = {x=-0.475, y=0.000, z=-1.584, rx=-0.000, ry=0.000, rz=-0.000, shoulder=lefty, elbow=epositive, wrist=wnegative, fatherId=fReference[0]}
  [212] = {x=-0.975, y=0.000, z=-1.591, rx=-0.000, ry=0.000, rz=-0.000, shoulder=lefty, elbow=epositive, wrist=wnegative, fatherId=fReference[0]}
  [213] = {x=-1.475, y=0.000, z=-1.599, rx=-0.000, ry=0.000, rz=-0.000, shoulder=lefty, elbow=epositive, wrist=wnegative, fatherId=fReference[0]}
  [214] = {x=-1.975, y=0.000, z=-1.607, rx=-0.000, ry=0.000, rz=-0.000, shoulder=lefty, elbow=epositive, wrist=wnegative, fatherId=fReference[0]}
  [215] = {x=-2.475, y=0.000, z=-1.615, rx=-0.000, ry=0.000, rz=-0.000, shoulder=lefty, elbow=epositive, wrist=wnegative, fatherId=fReference[0]}
  [216] = {x=-2.975, y=0.000, z=-1.623, rx=-0.000, ry=0.000, rz=-0.000, shoulder=lefty, elbow=epositive, wrist=wnegative, fatherId=fReference[0]}
  [217] = {x=-3.474, y=0.000, z=-1.630, rx=-0.000, ry=0.000, rz=-0.000, shoulder=lefty, elbow=epositive, wrist=wnegative, fatherId=fReference[0]}
  [218] = {x=-3.974, y=0.000, z=-1.638, rx=-0.000, ry=0.000, rz=-0.000, shoulder=lefty, elbow=epositive, wrist=wnegative, fatherId=fReference[0]}
  [219] = {x=-4.474, y=0.000, z=-1.646, rx=-0.000, ry=0.000, rz=-0.000, shoulder=lefty, elbow=epositive, wrist=wnegative, fatherId=fReference[0]}
  [220] = {x=-4.974, y=0.000, z=-1.654, rx=-0.000, ry=0.000, rz=-0.000, shoulder=lefty, elbow=epositive, wrist=wnegative, fatherId=fReference[0]}
  [221] = {x=-5.474, y=0.000, z=-1.662, rx=-0.000, ry=0.000, rz=-0.000, shoulder=lefty, elbow=epositive, wrist=wnegative, fatherId=fReference[0]}
  [222] = {x=-5.973, y=0.000, z=-1.670, rx=-0.000, ry=0.000, rz=-0.000, shoulder=lefty, elbow=epositive, wrist=wnegative, fatherId=fReference[0]}
  [223] = {x=-6.473, y=0.000, z=-1.678, rx=-0.000, ry=0.000, rz=-0.000, shoulder=lefty, elbow=epositive, wrist=wnegative, fatherId=fReference[0]}
  [224] = {x=-6.973, y=0.000, z=-1.686, rx=-0.000, ry=0.000, rz=-0.000, shoulder=lefty, elbow=epositive, wrist=wnegative, fatherId=fReference[0]}
  [225] = {x=-7.473, y=0.000, z=-1.694, rx=-0.000, ry=0.000, rz=-0.000, shoulder=lefty, elbow=epositive, wrist=wnegative, fatherId=fReference[0]}
  [226] = {x=-7.973, y=0.000, z=-1.702, rx=-0.000, ry=0.000, rz=-0.000, shoulder=lefty, elbow=epositive, wrist=wnegative, fatherId=fReference[0]}
  [227] = {x=-8.473, y=0.000, z=-1.710, rx=-0.000, ry=0.000, rz=-0.000, shoulder=lefty, elbow=epositive, wrist=wnegative, fatherId=fReference[0]}
  [228] = {x=-8.972, y=0.000, z=-1.718, rx=-0.000, ry=0.000, rz=-0.000, shoulder=lefty, elbow=epositive, wrist=wnegative, fatherId=fReference[0]}
  [229] = {x=-9.472, y=0.000, z=-1.726, rx=-0.000, ry=0.000, rz=-0.000, shoulder=lefty, elbow=epositive, wrist=wnegative, fatherId=fReference[0]}
  [230] = {x=-9.972, y=0.000, z=-1.734, rx=-0.000, ry=0.000, rz=-0.000, shoulder=lefty, elbow=epositive, wrist=wnegative, fatherId=fReference[0]}
  [231] = {x=-10.472, y=0.000, z=-1.742, rx=-0.000, ry=0.000, rz=-0.000, shoulder=lefty, elbow=epositive, wrist=wnegative, fatherId=fReference[0]}
  [232] = {x=-10.972, y=0.000, z=-1.750, rx=-0.000, ry=0.000, rz=-0.000, shoulder=lefty, elbow=epositive, wrist=wnegative, fatherId=fReference[0]}
  [233] = {x=-11.471, y=0.000, z=-1.758, rx=-0.000, ry=0.000, rz=-0.000, shoulder=lefty, elbow=epositive, wrist=wnegative, fatherId=fReference[0]}
  [234] = {x=-11.971, y=0.000, z=-1.766, rx=-0.000, ry=0.000, rz=-0.000, shoulder=lefty, elbow=epositive, wrist=wnegative, fatherId=fReference[0]}
  [235] = {x=-12.471, y=0.000, z=-1.774, rx=-0.000, ry=0.000, rz=-0.000, shoulder=lefty, elbow=epositive, wrist=wnegative, fatherId=fReference[0]}
  [236] = {x=-12.971, y=0.000, z=-1.782, rx=-0.000, ry=0.000, rz=-0.000, shoulder=lefty, elbow=epositive, wrist=wnegative, fatherId=fReference[0]}
  [237] = {x=-13.471, y=0.000, z=-1.790, rx=-0.000, ry=0.000, rz=-0.000, shoulder=lefty, elbow=epositive, wrist=wnegative, fatherId=fReference[0]}
  [238] = {x=-13.970, y=0.000, z=-1.799, rx=-0.000, ry=0.000, rz=-0.000, shoulder=lefty, elbow=epositive, wrist=wnegative, fatherId=fReference[0]}
  [239] = {x=-14.470, y=0.000, z=-1.807, rx=-0.000, ry=0.000, rz=-0.000, shoulder=lefty, elbow=epositive, wrist=wnegative, fatherId=fReference[0]}
  [240] = {x=-14.970, y=0.000, z=-1.815, rx=-0.000, ry=0.000, rz=-0.000, shoulder=lefty, elbow=epositive, wrist=wnegative, fatherId=fReference[0]}
  [241] = {x=-15.470, y=0.000, z=-1.824, rx=-0.000, ry=0.000, rz=-0.000, shoulder=lefty, elbow=epositive, wrist=wnegative, fatherId=fReference[0]}
  [242] = {x=-15.969, y=0.000, z=-1.832, rx=-0.000, ry=0.000, rz=-0.000, shoulder=lefty, elbow=epositive, wrist=wnegative, fatherId=fReference[0]}
  [243] = {x=-16.469, y=0.000, z=-1.840, rx=-0.000, ry=0.000, rz=-0.000, shoulder=lefty, elbow=epositive, wrist=wnegative, fatherId=fReference[0]}
  [244] = {x=-16.969, y=0.000, z=-1.849, rx=-0.000, ry=0.000, rz=-0.000, shoulder=lefty, elbow=epositive, wrist=wnegative, fatherId=fReference[0]}
  [245] = {x=-17.469, y=0.000, z=-1.857, rx=-0.000, ry=0.000, rz=-0.000, shoulder=lefty, elbow=epositive, wrist=wnegative, fatherId=fReference[0]}
  [246] = {x=-17.968, y=0.000, z=-1.865, rx=-0.000, ry=0.000, rz=-0.000, shoulder=lefty, elbow=epositive, wrist=wnegative, fatherId=fReference[0]}
  [247] = {x=-18.468, y=0.000, z=-1.874, rx=-0.000, ry=0.000, rz=-0.000, shoulder=lefty, elbow=epositive, wrist=wnegative, fatherId=fReference[0]}
  [248] = {x=-18.968, y=0.000, z=-1.883, rx=-0.000, ry=0.000, rz=-0.000, shoulder=lefty, elbow=epositive, wrist=wnegative, fatherId=fReference[0]}
  [249] = {x=-19.467, y=0.000, z=-1.891, rx=-0.000, ry=0.000, rz=-0.000, shoulder=lefty, elbow=epositive, wrist=wnegative, fatherId=fReference[0]}
  [250] = {x=-19.967, y=0.000, z=-1.900, rx=-0.000, ry=0.000, rz=-0.000, shoulder=lefty, elbow=epositive, wrist=wnegative, fatherId=fReference[0]}
  [251] = {x=-20.466, y=0.000, z=-1.908, rx=-0.000, ry=0.000, rz=-0.000, shoulder=lefty, elbow=epositive, wrist=wnegative, fatherId=fReference[0]}
  [252] = {x=-20.966, y=0.000, z=-1.917, rx=-0.000, ry=0.000, rz=-0.000, shoulder=lefty, elbow=epositive, wrist=wnegative, fatherId=fReference[0]}
  [253] = {x=-21.466, y=0.000, z=-1.925, rx=-0.000, ry=0.000, rz=-0.000, shoulder=lefty, elbow=epositive, wrist=wnegative, fatherId=fReference[0]}
  [254] = {x=-21.965, y=0.000, z=-1.934, rx=-0.000, ry=0.000, rz=-0.000, shoulder=lefty, elbow=epositive, wrist=wnegative, fatherId=fReference[0]}
  [255] = {x=-22.465, y=0.000, z=-1.943, rx=-0.000, ry=0.000, rz=-0.000, shoulder=lefty, elbow=epositive, wrist=wnegative, fatherId=fReference[0]}
  [256] = {x=-22.965, y=0.000, z=-1.952, rx=-0.000, ry=0.000, rz=-0.000, shoulder=lefty, elbow=epositive, wrist=wnegative, fatherId=fReference[0]}
  [257] = {x=-23.464, y=0.000, z=-1.960, rx=-0.000, ry=0.000, rz=-0.000, shoulder=lefty, elbow=epositive, wrist=wnegative, fatherId=fReference[0]}
  [258] = {x=-23.964, y=0.000, z=-1.969, rx=-0.000, ry=0.000, rz=-0.000, shoulder=lefty, elbow=epositive, wrist=wnegative, fatherId=fReference[0]}
  [259] = {x=-24.464, y=0.000, z=-1.978, rx=-0.000, ry=0.000, rz=-0.000, shoulder=lefty, elbow=epositive, wrist=wnegative, fatherId=fReference[0]}
  [260] = {x=-24.963, y=0.000, z=-1.987, rx=-0.000, ry=0.000, rz=-0.000, shoulder=lefty, elbow=epositive, wrist=wnegative, fatherId=fReference[0]}
  [261] = {x=-25.463, y=0.000, z=-1.996, rx=-0.000, ry=0.000, rz=-0.000, shoulder=lefty, elbow=epositive, wrist=wnegative, fatherId=fReference[0]}
  [262] = {x=-25.962, y=0.000, z=-2.005, rx=-0.000, ry=0.000, rz=-0.000, shoulder=lefty, elbow=epositive, wrist=wnegative, fatherId=fReference[0]}
  [263] = {x=-26.462, y=0.000, z=-2.014, rx=-0.000, ry=0.000, rz=-0.000, shoulder=lefty, elbow=epositive, wrist=wnegative, fatherId=fReference[0]}
  [264] = {x=-26.962, y=0.000, z=-2.023, rx=-0.000, ry=0.000, rz=-0.000, shoulder=lefty, elbow=epositive, wrist=wnegative, fatherId=fReference[0]}
  [265] = {x=-27.461, y=0.000, z=-2.032, rx=-0.000, ry=0.000, rz=-0.000, shoulder=lefty, elbow=epositive, wrist=wnegative, fatherId=fReference[0]}
  [266] = {x=-27.961, y=0.000, z=-2.041, rx=-0.000, ry=0.000, rz=-0.000, shoulder=lefty, elbow=epositive, wrist=wnegative, fatherId=fReference[0]}
  [267] = {x=-28.461, y=0.000, z=-2.050, rx=-0.000, ry=0.000, rz=-0.000, shoulder=lefty, elbow=epositive, wrist=wnegative, fatherId=fReference[0]}
  [268] = {x=-28.960, y=0.000, z=-2.059, rx=-0.000, ry=0.000, rz=-0.000, shoulder=lefty, elbow=epositive, wrist=wnegative, fatherId=fReference[0]}
  [269] = {x=-29.460, y=0.000, z=-2.069, rx=-0.000, ry=0.000, rz=-0.000, shoulder=lefty, elbow=epositive, wrist=wnegative, fatherId=fReference[0]}
  [270] = {x=-29.960, y=0.000, z=-2.078, rx=-0.000, ry=0.000, rz=-0.000, shoulder=lefty, elbow=epositive, wrist=wnegative, fatherId=fReference[0]}
  [271] = {x=-30.459, y=0.000, z=-2.087, rx=-0.000, ry=0.000, rz=-0.000, shoulder=lefty, elbow=epositive, wrist=wnegative, fatherId=fReference[0]}
  [272] = {x=-30.959, y=0.000, z=-2.097, rx=-0.000, ry=0.000, rz=-0.000, shoulder=lefty, elbow=epositive, wrist=wnegative, fatherId=fReference[0]}
  [273] = {x=-31.458, y=0.000, z=-2.107, rx=-0.000, ry=0.000, rz=-0.000, shoulder=lefty, elbow=epositive, wrist=wnegative, fatherId=fReference[0]}
  [274] = {x=-31.958, y=0.000, z=-2.116, rx=-0.000, ry=0.000, rz=-0.000, shoulder=lefty, elbow=epositive, wrist=wnegative, fatherId=fReference[0]}
  [275] = {x=-32.458, y=0.000, z=-2.125, rx=-0.000, ry=0.000, rz=-0.000, shoulder=lefty, elbow=epositive, wrist=wnegative, fatherId=fReference[0]}
  [276] = {x=-32.958, y=0.000, z=-2.135, rx=-0.000, ry=0.000, rz=-0.000, shoulder=lefty, elbow=epositive, wrist=wnegative, fatherId=fReference[0]}
  [277] = {x=-33.458, y=0.000, z=-2.144, rx=-0.000, ry=0.000, rz=-0.000, shoulder=lefty, elbow=epositive, wrist=wnegative, fatherId=fReference[0]}
  [278] = {x=-33.918, y=0.000, z=-2.146, rx=-0.000, ry=0.000, rz=-0.000, shoulder=lefty, elbow=epositive, wrist=wnegative, fatherId=fReference[0]}
  [279] = {x=-33.419, y=0.000, z=-2.150, rx=-0.000, ry=0.000, rz=-0.000, shoulder=lefty, elbow=epositive, wrist=wnegative, fatherId=fReference[0]}
  [280] = {x=-32.919, y=0.000, z=-2.155, rx=-0.000, ry=0.000, rz=-0.000, shoulder=lefty, elbow=epositive, wrist=wnegative, fatherId=fReference[0]}
  [281] = {x=-32.419, y=0.000, z=-2.160, rx=-0.000, ry=0.000, rz=-0.000, shoulder=lefty, elbow=epositive, wrist=wnegative, fatherId=fReference[0]}
  [282] = {x=-31.920, y=0.000, z=-2.166, rx=-0.000, ry=0.000, rz=-0.000, shoulder=lefty, elbow=epositive, wrist=wnegative, fatherId=fReference[0]}
  [283] = {x=-31.420, y=0.000, z=-2.171, rx=-0.000, ry=0.000, rz=-0.000, shoulder=lefty, elbow=epositive, wrist=wnegative, fatherId=fReference[0]}
  [284] = {x=-30.920, y=0.000, z=-2.178, rx=-0.000, ry=0.000, rz=-0.000, shoulder=lefty, elbow=epositive, wrist=wnegative, fatherId=fReference[0]}
  [285] = {x=-30.421, y=0.000, z=-2.184, rx=-0.000, ry=0.000, rz=-0.000, shoulder=lefty, elbow=epositive, wrist=wnegative, fatherId=fReference[0]}
  [286] = {x=-29.921, y=0.000, z=-2.190, rx=-0.000, ry=0.000, rz=-0.000, shoulder=lefty, elbow=epositive, wrist=wnegative, fatherId=fReference[0]}
  [287] = {x=-29.421, y=0.000, z=-2.197, rx=-0.000, ry=0.000, rz=-0.000, shoulder=lefty, elbow=epositive, wrist=wnegative, fatherId=fReference[0]}
  [288] = {x=-28.921, y=0.000, z=-2.204, rx=-0.000, ry=0.000, rz=-0.000, shoulder=lefty, elbow=epositive, wrist=wnegative, fatherId=fReference[0]}
  [289] = {x=-28.421, y=0.000, z=-2.210, rx=-0.000, ry=0.000, rz=-0.000, shoulder=lefty, elbow=epositive, wrist=wnegative, fatherId=fReference[0]}
  [290] = {x=-27.921, y=0.000, z=-2.217, rx=-0.000, ry=0.000, rz=-0.000, shoulder=lefty, elbow=epositive, wrist=wnegative, fatherId=fReference[0]}
  [291] = {x=-27.421, y=0.000, z=-2.224, rx=-0.000, ry=0.000, rz=-0.000, shoulder=lefty, elbow=epositive, wrist=wnegative, fatherId=fReference[0]}
  [292] = {x=-26.921, y=0.000, z=-2.231, rx=-0.000, ry=0.000, rz=-0.000, shoulder=lefty, elbow=epositive, wrist=wnegative, fatherId=fReference[0]}
  [293] = {x=-26.421, y=0.000, z=-2.238, rx=-0.000, ry=0.000, rz=-0.000, shoulder=lefty, elbow=epositive, wrist=wnegative, fatherId=fReference[0]}
  [294] = {x=-25.921, y=0.000, z=-2.245, rx=-0.000, ry=0.000, rz=-0.000, shoulder=lefty, elbow=epositive, wrist=wnegative, fatherId=fReference[0]}
  [295] = {x=-25.421, y=0.000, z=-2.252, rx=-0.000, ry=0.000, rz=-0.000, shoulder=lefty, elbow=epositive, wrist=wnegative, fatherId=fReference[0]}
  [296] = {x=-24.921, y=0.000, z=-2.260, rx=-0.000, ry=0.000, rz=-0.000, shoulder=lefty, elbow=epositive, wrist=wnegative, fatherId=fReference[0]}
  [297] = {x=-24.421, y=0.000, z=-2.267, rx=-0.000, ry=0.000, rz=-0.000, shoulder=lefty, elbow=epositive, wrist=wnegative, fatherId=fReference[0]}
  [298] = {x=-23.921, y=0.000, z=-2.274, rx=-0.000, ry=0.000, rz=-0.000, shoulder=lefty, elbow=epositive, wrist=wnegative, fatherId=fReference[0]}
  [299] = {x=-23.420, y=0.000, z=-2.281, rx=-0.000, ry=0.000, rz=-0.000, shoulder=lefty, elbow=epositive, wrist=wnegative, fatherId=fReference[0]}
  [300] = {x=-22.920, y=0.000, z=-2.289, rx=-0.000, ry=0.000, rz=-0.000, shoulder=lefty, elbow=epositive, wrist=wnegative, fatherId=fReference[0]}
  [301] = {x=-22.420, y=0.000, z=-2.296, rx=-0.000, ry=0.000, rz=-0.000, shoulder=lefty, elbow=epositive, wrist=wnegative, fatherId=fReference[0]}
  [302] = {x=-21.920, y=0.000, z=-2.304, rx=-0.000, ry=0.000, rz=-0.000, shoulder=lefty, elbow=epositive, wrist=wnegative, fatherId=fReference[0]}
  [303] = {x=-21.420, y=0.000, z=-2.311, rx=-0.000, ry=0.000, rz=-0.000, shoulder=lefty, elbow=epositive, wrist=wnegative, fatherId=fReference[0]}
  [304] = {x=-20.920, y=0.000, z=-2.318, rx=-0.000, ry=0.000, rz=-0.000, shoulder=lefty, elbow=epositive, wrist=wnegative, fatherId=fReference[0]}
  [305] = {x=-20.420, y=0.000, z=-2.326, rx=-0.000, ry=0.000, rz=-0.000, shoulder=lefty, elbow=epositive, wrist=wnegative, fatherId=fReference[0]}
  [306] = {x=-19.920, y=0.000, z=-2.333, rx=-0.000, ry=0.000, rz=-0.000, shoulder=lefty, elbow=epositive, wrist=wnegative, fatherId=fReference[0]}
  [307] = {x=-19.419, y=0.000, z=-2.341, rx=-0.000, ry=0.000, rz=-0.000, shoulder=lefty, elbow=epositive, wrist=wnegative, fatherId=fReference[0]}
  [308] = {x=-18.919, y=0.000, z=-2.348, rx=-0.000, ry=0.000, rz=-0.000, shoulder=lefty, elbow=epositive, wrist=wnegative, fatherId=fReference[0]}
  [309] = {x=-18.419, y=0.000, z=-2.356, rx=-0.000, ry=0.000, rz=-0.000, shoulder=lefty, elbow=epositive, wrist=wnegative, fatherId=fReference[0]}
  [310] = {x=-17.919, y=0.000, z=-2.363, rx=-0.000, ry=0.000, rz=-0.000, shoulder=lefty, elbow=epositive, wrist=wnegative, fatherId=fReference[0]}
  [311] = {x=-17.418, y=0.000, z=-2.371, rx=-0.000, ry=0.000, rz=-0.000, shoulder=lefty, elbow=epositive, wrist=wnegative, fatherId=fReference[0]}
  [312] = {x=-16.918, y=0.000, z=-2.378, rx=-0.000, ry=0.000, rz=-0.000, shoulder=lefty, elbow=epositive, wrist=wnegative, fatherId=fReference[0]}
  [313] = {x=-16.418, y=0.000, z=-2.386, rx=-0.000, ry=0.000, rz=-0.000, shoulder=lefty, elbow=epositive, wrist=wnegative, fatherId=fReference[0]}
  [314] = {x=-15.918, y=0.000, z=-2.393, rx=-0.000, ry=0.000, rz=-0.000, shoulder=lefty, elbow=epositive, wrist=wnegative, fatherId=fReference[0]}
  [315] = {x=-15.417, y=0.000, z=-2.401, rx=-0.000, ry=0.000, rz=-0.000, shoulder=lefty, elbow=epositive, wrist=wnegative, fatherId=fReference[0]}
  [316] = {x=-14.917, y=0.000, z=-2.408, rx=-0.000, ry=0.000, rz=-0.000, shoulder=lefty, elbow=epositive, wrist=wnegative, fatherId=fReference[0]}
  [317] = {x=-14.417, y=0.000, z=-2.416, rx=-0.000, ry=0.000, rz=-0.000, shoulder=lefty, elbow=epositive, wrist=wnegative, fatherId=fReference[0]}
  [318] = {x=-13.916, y=0.000, z=-2.424, rx=-0.000, ry=0.000, rz=-0.000, shoulder=lefty, elbow=epositive, wrist=wnegative, fatherId=fReference[0]}
  [319] = {x=-13.416, y=0.000, z=-2.431, rx=-0.000, ry=0.000, rz=-0.000, shoulder=lefty, elbow=epositive, wrist=wnegative, fatherId=fReference[0]}
  [320] = {x=-12.916, y=0.000, z=-2.439, rx=-0.000, ry=0.000, rz=-0.000, shoulder=lefty, elbow=epositive, wrist=wnegative, fatherId=fReference[0]}
  [321] = {x=-12.415, y=0.000, z=-2.446, rx=-0.000, ry=0.000, rz=-0.000, shoulder=lefty, elbow=epositive, wrist=wnegative, fatherId=fReference[0]}
  [322] = {x=-11.915, y=0.000, z=-2.454, rx=-0.000, ry=0.000, rz=-0.000, shoulder=lefty, elbow=epositive, wrist=wnegative, fatherId=fReference[0]}
  [323] = {x=-11.415, y=0.000, z=-2.462, rx=-0.000, ry=0.000, rz=-0.000, shoulder=lefty, elbow=epositive, wrist=wnegative, fatherId=fReference[0]}
  [324] = {x=-10.914, y=0.000, z=-2.469, rx=-0.000, ry=0.000, rz=-0.000, shoulder=lefty, elbow=epositive, wrist=wnegative, fatherId=fReference[0]}
  [325] = {x=-10.414, y=0.000, z=-2.477, rx=-0.000, ry=0.000, rz=-0.000, shoulder=lefty, elbow=epositive, wrist=wnegative, fatherId=fReference[0]}
  [326] = {x=-9.914, y=0.000, z=-2.485, rx=-0.000, ry=0.000, rz=-0.000, shoulder=lefty, elbow=epositive, wrist=wnegative, fatherId=fReference[0]}
  [327] = {x=-9.413, y=0.000, z=-2.492, rx=-0.000, ry=0.000, rz=-0.000, shoulder=lefty, elbow=epositive, wrist=wnegative, fatherId=fReference[0]}
  [328] = {x=-8.913, y=0.000, z=-2.500, rx=-0.000, ry=0.000, rz=-0.000, shoulder=lefty, elbow=epositive, wrist=wnegative, fatherId=fReference[0]}
  [329] = {x=-8.413, y=0.000, z=-2.508, rx=-0.000, ry=0.000, rz=-0.000, shoulder=lefty, elbow=epositive, wrist=wnegative, fatherId=fReference[0]}
  [330] = {x=-7.912, y=0.000, z=-2.515, rx=-0.000, ry=0.000, rz=-0.000, shoulder=lefty, elbow=epositive, wrist=wnegative, fatherId=fReference[0]}
  [331] = {x=-7.412, y=0.000, z=-2.523, rx=-0.000, ry=0.000, rz=-0.000, shoulder=lefty, elbow=epositive, wrist=wnegative, fatherId=fReference[0]}
  [332] = {x=-6.911, y=0.000, z=-2.531, rx=-0.000, ry=0.000, rz=-0.000, shoulder=lefty, elbow=epositive, wrist=wnegative, fatherId=fReference[0]}
  [333] = {x=-6.411, y=0.000, z=-2.539, rx=-0.000, ry=0.000, rz=-0.000, shoulder=lefty, elbow=epositive, wrist=wnegative, fatherId=fReference[0]}
  [334] = {x=-5.910, y=0.000, z=-2.546, rx=-0.000, ry=0.000, rz=-0.000, shoulder=lefty, elbow=epositive, wrist=wnegative, fatherId=fReference[0]}
  [335] = {x=-5.410, y=0.000, z=-2.554, rx=-0.000, ry=0.000, rz=-0.000, shoulder=lefty, elbow=epositive, wrist=wnegative, fatherId=fReference[0]}
  [336] = {x=-4.909, y=0.000, z=-2.562, rx=-0.000, ry=0.000, rz=-0.000, shoulder=lefty, elbow=epositive, wrist=wnegative, fatherId=fReference[0]}
  [337] = {x=-4.409, y=0.000, z=-2.570, rx=-0.000, ry=0.000, rz=-0.000, shoulder=lefty, elbow=epositive, wrist=wnegative, fatherId=fReference[0]}
  [338] = {x=-3.909, y=0.000, z=-2.578, rx=-0.000, ry=0.000, rz=-0.000, shoulder=lefty, elbow=epositive, wrist=wnegative, fatherId=fReference[0]}
  [339] = {x=-3.408, y=0.000, z=-2.586, rx=-0.000, ry=0.000, rz=-0.000, shoulder=lefty, elbow=epositive, wrist=wnegative, fatherId=fReference[0]}
  [340] = {x=-2.908, y=0.000, z=-2.594, rx=-0.000, ry=0.000, rz=-0.000, shoulder=lefty, elbow=epositive, wrist=wnegative, fatherId=fReference[0]}
  [341] = {x=-2.407, y=0.000, z=-2.602, rx=-0.000, ry=0.000, rz=-0.000, shoulder=lefty, elbow=epositive, wrist=wnegative, fatherId=fReference[0]}
  [342] = {x=-1.907, y=0.000, z=-2.610, rx=-0.000, ry=0.000, rz=-0.000, shoulder=lefty, elbow=epositive, wrist=wnegative, fatherId=fReference[0]}
  [343] = {x=-1.406, y=0.000, z=-2.617, rx=-0.000, ry=0.000, rz=-0.000, shoulder=lefty, elbow=epositive, wrist=wnegative, fatherId=fReference[0]}
  [344] = {x=-0.905, y=0.000, z=-2.626, rx=-0.000, ry=0.000, rz=-0.000, shoulder=lefty, elbow=epositive, wrist=wnegative, fatherId=fReference[0]}
  [345] = {x=-0.405, y=0.000, z=-2.634, rx=-0.000, ry=0.000, rz=-0.000, shoulder=lefty, elbow=epositive, wrist=wnegative, fatherId=fReference[0]}
  [346] = {x=0.096, y=0.000, z=-2.642, rx=-0.000, ry=0.000, rz=-0.000, shoulder=lefty, elbow=epositive, wrist=wnegative, fatherId=fReference[0]}
  [347] = {x=0.596, y=0.000, z=-2.650, rx=-0.000, ry=0.000, rz=-0.000, shoulder=lefty, elbow=epositive, wrist=wnegative, fatherId=fReference[0]}
  [348] = {x=1.097, y=0.000, z=-2.658, rx=-0.000, ry=0.000, rz=-0.000, shoulder=lefty, elbow=epositive, wrist=wnegative, fatherId=fReference[0]}
  [349] = {x=1.598, y=0.000, z=-2.666, rx=-0.000, ry=0.000, rz=-0.000, shoulder=lefty, elbow=epositive, wrist=wnegative, fatherId=fReference[0]}
  [350] = {x=2.099, y=0.000, z=-2.674, rx=-0.000, ry=0.000, rz=-0.000, shoulder=lefty, elbow=epositive, wrist=wnegative, fatherId=fReference[0]}
  [351] = {x=2.600, y=0.000, z=-2.683, rx=-0.000, ry=0.000, rz=-0.000, shoulder=lefty, elbow=epositive, wrist=wnegative, fatherId=fReference[0]}
  [352] = {x=3.100, y=0.000, z=-2.691, rx=-0.000, ry=0.000, rz=-0.000, shoulder=lefty, elbow=epositive, wrist=wnegative, fatherId=fReference[0]}
  [353] = {x=3.601, y=0.000, z=-2.699, rx=-0.000, ry=0.000, rz=-0.000, shoulder=lefty, elbow=epositive, wrist=wnegative, fatherId=fReference[0]}
  [354] = {x=4.102, y=0.000, z=-2.708, rx=-0.000, ry=0.000, rz=-0.000, shoulder=lefty, elbow=epositive, wrist=wnegative, fatherId=fReference[0]}
  [355] = {x=4.603, y=0.000, z=-2.716, rx=-0.000, ry=0.000, rz=-0.000, shoulder=lefty, elbow=epositive, wrist=wnegative, fatherId=fReference[0]}
  [356] = {x=5.104, y=0.000, z=-2.724, rx=-0.000, ry=0.000, rz=-0.000, shoulder=lefty, elbow=epositive, wrist=wnegative, fatherId=fReference[0]}
  [357] = {x=5.604, y=0.000, z=-2.733, rx=-0.000, ry=0.000, rz=-0.000, shoulder=lefty, elbow=epositive, wrist=wnegative, fatherId=fReference[0]}
  [358] = {x=6.105, y=0.000, z=-2.741, rx=-0.000, ry=0.000, rz=-0.000, shoulder=lefty, elbow=epositive, wrist=wnegative, fatherId=fReference[0]}
  [359] = {x=6.606, y=0.000, z=-2.749, rx=-0.000, ry=0.000, rz=-0.000, shoulder=lefty, elbow=epositive, wrist=wnegative, fatherId=fReference[0]}
  [360] = {x=7.107, y=0.000, z=-2.758, rx=-0.000, ry=0.000, rz=-0.000, shoulder=lefty, elbow=epositive, wrist=wnegative, fatherId=fReference[0]}
  [361] = {x=7.608, y=0.000, z=-2.766, rx=-0.000, ry=0.000, rz=-0.000, shoulder=lefty, elbow=epositive, wrist=wnegative, fatherId=fReference[0]}
  [362] = {x=8.109, y=0.000, z=-2.775, rx=-0.000, ry=0.000, rz=-0.000, shoulder=lefty, elbow=epositive, wrist=wnegative, fatherId=fReference[0]}
  [363] = {x=8.610, y=0.000, z=-2.783, rx=-0.000, ry=0.000, rz=-0.000, shoulder=lefty, elbow=epositive, wrist=wnegative, fatherId=fReference[0]}
  [364] = {x=9.111, y=0.000, z=-2.792, rx=-0.000, ry=0.000, rz=-0.000, shoulder=lefty, elbow=epositive, wrist=wnegative, fatherId=fReference[0]}
  [365] = {x=9.612, y=0.000, z=-2.800, rx=-0.000, ry=0.000, rz=-0.000, shoulder=lefty, elbow=epositive, wrist=wnegative, fatherId=fReference[0]}
  [366] = {x=10.113, y=0.000, z=-2.809, rx=-0.000, ry=0.000, rz=-0.000, shoulder=lefty, elbow=epositive, wrist=wnegative, fatherId=fReference[0]}
  [367] = {x=10.614, y=0.000, z=-2.817, rx=-0.000, ry=0.000, rz=-0.000, shoulder=lefty, elbow=epositive, wrist=wnegative, fatherId=fReference[0]}
  [368] = {x=11.115, y=0.000, z=-2.826, rx=-0.000, ry=0.000, rz=-0.000, shoulder=lefty, elbow=epositive, wrist=wnegative, fatherId=fReference[0]}
  [369] = {x=11.616, y=0.000, z=-2.835, rx=-0.000, ry=0.000, rz=-0.000, shoulder=lefty, elbow=epositive, wrist=wnegative, fatherId=fReference[0]}
  [370] = {x=12.117, y=0.000, z=-2.843, rx=-0.000, ry=0.000, rz=-0.000, shoulder=lefty, elbow=epositive, wrist=wnegative, fatherId=fReference[0]}
  [371] = {x=12.618, y=0.000, z=-2.852, rx=-0.000, ry=0.000, rz=-0.000, shoulder=lefty, elbow=epositive, wrist=wnegative, fatherId=fReference[0]}
  [372] = {x=13.120, y=0.000, z=-2.861, rx=-0.000, ry=0.000, rz=-0.000, shoulder=lefty, elbow=epositive, wrist=wnegative, fatherId=fReference[0]}
  [373] = {x=13.621, y=0.000, z=-2.869, rx=-0.000, ry=0.000, rz=-0.000, shoulder=lefty, elbow=epositive, wrist=wnegative, fatherId=fReference[0]}
  [374] = {x=14.122, y=0.000, z=-2.878, rx=-0.000, ry=0.000, rz=-0.000, shoulder=lefty, elbow=epositive, wrist=wnegative, fatherId=fReference[0]}
  [375] = {x=14.623, y=0.000, z=-2.887, rx=-0.000, ry=0.000, rz=-0.000, shoulder=lefty, elbow=epositive, wrist=wnegative, fatherId=fReference[0]}
  [376] = {x=15.124, y=0.000, z=-2.896, rx=-0.000, ry=0.000, rz=-0.000, shoulder=lefty, elbow=epositive, wrist=wnegative, fatherId=fReference[0]}
  [377] = {x=15.626, y=0.000, z=-2.904, rx=-0.000, ry=0.000, rz=-0.000, shoulder=lefty, elbow=epositive, wrist=wnegative, fatherId=fReference[0]}
  [378] = {x=16.127, y=0.000, z=-2.913, rx=-0.000, ry=0.000, rz=-0.000, shoulder=lefty, elbow=epositive, wrist=wnegative, fatherId=fReference[0]}
  [379] = {x=16.629, y=0.000, z=-2.922, rx=-0.000, ry=0.000, rz=-0.000, shoulder=lefty, elbow=epositive, wrist=wnegative, fatherId=fReference[0]}
  [380] = {x=17.130, y=0.000, z=-2.931, rx=-0.000, ry=0.000, rz=-0.000, shoulder=lefty, elbow=epositive, wrist=wnegative, fatherId=fReference[0]}
  [381] = {x=17.631, y=0.000, z=-2.940, rx=-0.000, ry=0.000, rz=-0.000, shoulder=lefty, elbow=epositive, wrist=wnegative, fatherId=fReference[0]}
  [382] = {x=18.133, y=0.000, z=-2.948, rx=-0.000, ry=0.000, rz=-0.000, shoulder=lefty, elbow=epositive, wrist=wnegative, fatherId=fReference[0]}
  [383] = {x=18.634, y=0.000, z=-2.957, rx=-0.000, ry=0.000, rz=-0.000, shoulder=lefty, elbow=epositive, wrist=wnegative, fatherId=fReference[0]}
  [384] = {x=19.136, y=0.000, z=-2.966, rx=-0.000, ry=0.000, rz=-0.000, shoulder=lefty, elbow=epositive, wrist=wnegative, fatherId=fReference[0]}
  [385] = {x=19.637, y=0.000, z=-2.975, rx=-0.000, ry=0.000, rz=-0.000, shoulder=lefty, elbow=epositive, wrist=wnegative, fatherId=fReference[0]}
  [386] = {x=20.139, y=0.000, z=-2.984, rx=-0.000, ry=0.000, rz=-0.000, shoulder=lefty, elbow=epositive, wrist=wnegative, fatherId=fReference[0]}
  [387] = {x=20.640, y=0.000, z=-2.993, rx=-0.000, ry=0.000, rz=-0.000, shoulder=lefty, elbow=epositive, wrist=wnegative, fatherId=fReference[0]}
  [388] = {x=21.142, y=0.000, z=-3.002, rx=-0.000, ry=0.000, rz=-0.000, shoulder=lefty, elbow=epositive, wrist=wnegative, fatherId=fReference[0]}
  [389] = {x=21.644, y=0.000, z=-3.011, rx=-0.000, ry=0.000, rz=-0.000, shoulder=lefty, elbow=epositive, wrist=wnegative, fatherId=fReference[0]}
  [390] = {x=22.146, y=0.000, z=-3.021, rx=-0.000, ry=0.000, rz=-0.000, shoulder=lefty, elbow=epositive, wrist=wnegative, fatherId=fReference[0]}
  [391] = {x=22.648, y=0.000, z=-3.030, rx=-0.000, ry=0.000, rz=-0.000, shoulder=lefty, elbow=epositive, wrist=wnegative, fatherId=fReference[0]}
  [392] = {x=23.150, y=0.000, z=-3.039, rx=-0.000, ry=0.000, rz=-0.000, shoulder=lefty, elbow=epositive, wrist=wnegative, fatherId=fReference[0]}
  [393] = {x=23.651, y=0.000, z=-3.048, rx=-0.000, ry=0.000, rz=-0.000, shoulder=lefty, elbow=epositive, wrist=wnegative, fatherId=fReference[0]}
  [394] = {x=24.153, y=0.000, z=-3.057, rx=-0.000, ry=0.000, rz=-0.000, shoulder=lefty, elbow=epositive, wrist=wnegative, fatherId=fReference[0]}
  [395] = {x=24.655, y=0.000, z=-3.066, rx=-0.000, ry=0.000, rz=-0.000, shoulder=lefty, elbow=epositive, wrist=wnegative, fatherId=fReference[0]}
  [396] = {x=25.157, y=0.000, z=-3.075, rx=-0.000, ry=0.000, rz=-0.000, shoulder=lefty, elbow=epositive, wrist=wnegative, fatherId=fReference[0]}
  [397] = {x=25.659, y=0.000, z=-3.084, rx=-0.000, ry=0.000, rz=-0.000, shoulder=lefty, elbow=epositive, wrist=wnegative, fatherId=fReference[0]}
  [398] = {x=26.161, y=0.000, z=-3.094, rx=-0.000, ry=0.000, rz=-0.000, shoulder=lefty, elbow=epositive, wrist=wnegative, fatherId=fReference[0]}
  [399] = {x=26.663, y=0.000, z=-3.103, rx=-0.000, ry=0.000, rz=-0.000, shoulder=lefty, elbow=epositive, wrist=wnegative, fatherId=fReference[0]}
  [400] = {x=27.165, y=0.000, z=-3.113, rx=-0.000, ry=0.000, rz=-0.000, shoulder=lefty, elbow=epositive, wrist=wnegative, fatherId=fReference[0]}
  [401] = {x=27.668, y=0.000, z=-3.123, rx=-0.000, ry=0.000, rz=-0.000, shoulder=lefty, elbow=epositive, wrist=wnegative, fatherId=fReference[0]}
  [402] = {x=28.170, y=0.000, z=-3.132, rx=-0.000, ry=0.000, rz=-0.000, shoulder=lefty, elbow=epositive, wrist=wnegative, fatherId=fReference[0]}
  [403] = {x=28.672, y=0.000, z=-3.142, rx=-0.000, ry=0.000, rz=-0.000, shoulder=lefty, elbow=epositive, wrist=wnegative, fatherId=fReference[0]}
  [404] = {x=29.174, y=0.000, z=-3.152, rx=-0.000, ry=0.000, rz=-0.000, shoulder=lefty, elbow=epositive, wrist=wnegative, fatherId=fReference[0]}
  [405] = {x=29.677, y=0.000, z=-3.162, rx=-0.000, ry=0.000, rz=-0.000, shoulder=lefty, elbow=epositive, wrist=wnegative, fatherId=fReference[0]}
  [406] = {x=30.180, y=0.000, z=-3.172, rx=-0.000, ry=0.000, rz=-0.000, shoulder=lefty, elbow=epositive, wrist=wnegative, fatherId=fReference[0]}
  [407] = {x=30.682, y=0.000, z=-3.182, rx=-0.000, ry=0.000, rz=-0.000, shoulder=lefty, elbow=epositive, wrist=wnegative, fatherId=fReference[0]}
  [408] = {x=31.185, y=0.000, z=-3.192, rx=-0.000, ry=0.000, rz=-0.000, shoulder=lefty, elbow=epositive, wrist=wnegative, fatherId=fReference[0]}
  [409] = {x=31.688, y=0.000, z=-3.202, rx=-0.000, ry=0.000, rz=-0.000, shoulder=lefty, elbow=epositive, wrist=wnegative, fatherId=fReference[0]}
  [410] = {x=32.191, y=0.000, z=-3.213, rx=-0.000, ry=0.000, rz=-0.000, shoulder=lefty, elbow=epositive, wrist=wnegative, fatherId=fReference[0]}
  [411] = {x=32.695, y=0.000, z=-3.223, rx=-0.000, ry=0.000, rz=-0.000, shoulder=lefty, elbow=epositive, wrist=wnegative, fatherId=fReference[0]}
  [412] = {x=33.198, y=0.000, z=-3.233, rx=-0.000, ry=0.000, rz=-0.000, shoulder=lefty, elbow=epositive, wrist=wnegative, fatherId=fReference[0]}
  [413] = {x=33.702, y=0.000, z=-3.244, rx=-0.000, ry=0.000, rz=-0.000, shoulder=lefty, elbow=epositive, wrist=wnegative, fatherId=fReference[0]}
  [414] = {x=34.120, y=0.000, z=-3.242, rx=-0.000, ry=0.000, rz=-0.000, shoulder=lefty, elbow=epositive, wrist=wnegative, fatherId=fReference[0]}
  [415] = {x=33.607, y=0.000, z=-3.241, rx=-0.000, ry=0.000, rz=-0.000, shoulder=lefty, elbow=epositive, wrist=wnegative, fatherId=fReference[0]}
  [416] = {x=33.099, y=0.000, z=-3.241, rx=-0.000, ry=0.000, rz=-0.000, shoulder=lefty, elbow=epositive, wrist=wnegative, fatherId=fReference[0]}
  [417] = {x=32.593, y=0.000, z=-3.244, rx=-0.000, ry=0.000, rz=-0.000, shoulder=lefty, elbow=epositive, wrist=wnegative, fatherId=fReference[0]}
  [418] = {x=32.089, y=0.000, z=-3.248, rx=-0.000, ry=0.000, rz=-0.000, shoulder=lefty, elbow=epositive, wrist=wnegative, fatherId=fReference[0]}
  [419] = {x=31.586, y=0.000, z=-3.253, rx=-0.000, ry=0.000, rz=-0.000, shoulder=lefty, elbow=epositive, wrist=wnegative, fatherId=fReference[0]}
  [420] = {x=31.084, y=0.000, z=-3.259, rx=-0.000, ry=0.000, rz=-0.000, shoulder=lefty, elbow=epositive, wrist=wnegative, fatherId=fReference[0]}
  [421] = {x=30.583, y=0.000, z=-3.266, rx=-0.000, ry=0.000, rz=-0.000, shoulder=lefty, elbow=epositive, wrist=wnegative, fatherId=fReference[0]}
  [422] = {x=30.082, y=0.000, z=-3.273, rx=-0.000, ry=0.000, rz=-0.000, shoulder=lefty, elbow=epositive, wrist=wnegative, fatherId=fReference[0]}
  [423] = {x=29.581, y=0.000, z=-3.280, rx=-0.000, ry=0.000, rz=-0.000, shoulder=lefty, elbow=epositive, wrist=wnegative, fatherId=fReference[0]}
  [424] = {x=29.080, y=0.000, z=-3.288, rx=-0.000, ry=0.000, rz=-0.000, shoulder=lefty, elbow=epositive, wrist=wnegative, fatherId=fReference[0]}
  [425] = {x=28.580, y=0.000, z=-3.295, rx=-0.000, ry=0.000, rz=-0.000, shoulder=lefty, elbow=epositive, wrist=wnegative, fatherId=fReference[0]}
  [426] = {x=28.080, y=0.000, z=-3.303, rx=-0.000, ry=0.000, rz=-0.000, shoulder=lefty, elbow=epositive, wrist=wnegative, fatherId=fReference[0]}
  [427] = {x=27.580, y=0.000, z=-3.311, rx=-0.000, ry=0.000, rz=-0.000, shoulder=lefty, elbow=epositive, wrist=wnegative, fatherId=fReference[0]}
  [428] = {x=27.079, y=0.000, z=-3.319, rx=-0.000, ry=0.000, rz=-0.000, shoulder=lefty, elbow=epositive, wrist=wnegative, fatherId=fReference[0]}
  [429] = {x=26.579, y=0.000, z=-3.327, rx=-0.000, ry=0.000, rz=-0.000, shoulder=lefty, elbow=epositive, wrist=wnegative, fatherId=fReference[0]}
  [430] = {x=26.079, y=0.000, z=-3.335, rx=-0.000, ry=0.000, rz=-0.000, shoulder=lefty, elbow=epositive, wrist=wnegative, fatherId=fReference[0]}
  [431] = {x=25.579, y=0.000, z=-3.344, rx=-0.000, ry=0.000, rz=-0.000, shoulder=lefty, elbow=epositive, wrist=wnegative, fatherId=fReference[0]}
  [432] = {x=25.079, y=0.000, z=-3.352, rx=-0.000, ry=0.000, rz=-0.000, shoulder=lefty, elbow=epositive, wrist=wnegative, fatherId=fReference[0]}
  [433] = {x=24.580, y=0.000, z=-3.360, rx=-0.000, ry=0.000, rz=-0.000, shoulder=lefty, elbow=epositive, wrist=wnegative, fatherId=fReference[0]}
  [434] = {x=24.080, y=0.000, z=-3.369, rx=-0.000, ry=0.000, rz=-0.000, shoulder=lefty, elbow=epositive, wrist=wnegative, fatherId=fReference[0]}
  [435] = {x=23.580, y=0.000, z=-3.377, rx=-0.000, ry=0.000, rz=-0.000, shoulder=lefty, elbow=epositive, wrist=wnegative, fatherId=fReference[0]}
  [436] = {x=23.080, y=0.000, z=-3.386, rx=-0.000, ry=0.000, rz=-0.000, shoulder=lefty, elbow=epositive, wrist=wnegative, fatherId=fReference[0]}
  [437] = {x=22.580, y=0.000, z=-3.394, rx=-0.000, ry=0.000, rz=-0.000, shoulder=lefty, elbow=epositive, wrist=wnegative, fatherId=fReference[0]}
  [438] = {x=22.081, y=0.000, z=-3.402, rx=-0.000, ry=0.000, rz=-0.000, shoulder=lefty, elbow=epositive, wrist=wnegative, fatherId=fReference[0]}
  [439] = {x=21.581, y=0.000, z=-3.411, rx=-0.000, ry=0.000, rz=-0.000, shoulder=lefty, elbow=epositive, wrist=wnegative, fatherId=fReference[0]}
  [440] = {x=21.081, y=0.000, z=-3.419, rx=-0.000, ry=0.000, rz=-0.000, shoulder=lefty, elbow=epositive, wrist=wnegative, fatherId=fReference[0]}
  [441] = {x=20.581, y=0.000, z=-3.427, rx=-0.000, ry=0.000, rz=-0.000, shoulder=lefty, elbow=epositive, wrist=wnegative, fatherId=fReference[0]}
  [442] = {x=20.081, y=0.000, z=-3.435, rx=-0.000, ry=0.000, rz=-0.000, shoulder=lefty, elbow=epositive, wrist=wnegative, fatherId=fReference[0]}
  [443] = {x=19.581, y=0.000, z=-3.443, rx=-0.000, ry=0.000, rz=-0.000, shoulder=lefty, elbow=epositive, wrist=wnegative, fatherId=fReference[0]}
  [444] = {x=19.081, y=0.000, z=-3.451, rx=-0.000, ry=0.000, rz=-0.000, shoulder=lefty, elbow=epositive, wrist=wnegative, fatherId=fReference[0]}
  [445] = {x=18.581, y=0.000, z=-3.459, rx=-0.000, ry=0.000, rz=-0.000, shoulder=lefty, elbow=epositive, wrist=wnegative, fatherId=fReference[0]}
  [446] = {x=18.081, y=0.000, z=-3.467, rx=-0.000, ry=0.000, rz=-0.000, shoulder=lefty, elbow=epositive, wrist=wnegative, fatherId=fReference[0]}
  [447] = {x=17.580, y=0.000, z=-3.475, rx=-0.000, ry=0.000, rz=-0.000, shoulder=lefty, elbow=epositive, wrist=wnegative, fatherId=fReference[0]}
  [448] = {x=17.080, y=0.000, z=-3.483, rx=-0.000, ry=0.000, rz=-0.000, shoulder=lefty, elbow=epositive, wrist=wnegative, fatherId=fReference[0]}
  [449] = {x=16.580, y=0.000, z=-3.491, rx=-0.000, ry=0.000, rz=-0.000, shoulder=lefty, elbow=epositive, wrist=wnegative, fatherId=fReference[0]}
  [450] = {x=16.080, y=0.000, z=-3.499, rx=-0.000, ry=0.000, rz=-0.000, shoulder=lefty, elbow=epositive, wrist=wnegative, fatherId=fReference[0]}
  [451] = {x=15.580, y=0.000, z=-3.507, rx=-0.000, ry=0.000, rz=-0.000, shoulder=lefty, elbow=epositive, wrist=wnegative, fatherId=fReference[0]}
  [452] = {x=15.080, y=0.000, z=-3.515, rx=-0.000, ry=0.000, rz=-0.000, shoulder=lefty, elbow=epositive, wrist=wnegative, fatherId=fReference[0]}
  [453] = {x=14.579, y=0.000, z=-3.523, rx=-0.000, ry=0.000, rz=-0.000, shoulder=lefty, elbow=epositive, wrist=wnegative, fatherId=fReference[0]}
  [454] = {x=14.079, y=0.000, z=-3.531, rx=-0.000, ry=0.000, rz=-0.000, shoulder=lefty, elbow=epositive, wrist=wnegative, fatherId=fReference[0]}
  [455] = {x=13.579, y=0.000, z=-3.539, rx=-0.000, ry=0.000, rz=-0.000, shoulder=lefty, elbow=epositive, wrist=wnegative, fatherId=fReference[0]}
  [456] = {x=13.079, y=0.000, z=-3.547, rx=-0.000, ry=0.000, rz=-0.000, shoulder=lefty, elbow=epositive, wrist=wnegative, fatherId=fReference[0]}
  [457] = {x=12.578, y=0.000, z=-3.554, rx=-0.000, ry=0.000, rz=-0.000, shoulder=lefty, elbow=epositive, wrist=wnegative, fatherId=fReference[0]}
  [458] = {x=12.078, y=0.000, z=-3.562, rx=-0.000, ry=0.000, rz=-0.000, shoulder=lefty, elbow=epositive, wrist=wnegative, fatherId=fReference[0]}
  [459] = {x=11.578, y=0.000, z=-3.570, rx=-0.000, ry=0.000, rz=-0.000, shoulder=lefty, elbow=epositive, wrist=wnegative, fatherId=fReference[0]}
  [460] = {x=11.078, y=0.000, z=-3.578, rx=-0.000, ry=0.000, rz=-0.000, shoulder=lefty, elbow=epositive, wrist=wnegative, fatherId=fReference[0]}
  [461] = {x=10.577, y=0.000, z=-3.586, rx=-0.000, ry=0.000, rz=-0.000, shoulder=lefty, elbow=epositive, wrist=wnegative, fatherId=fReference[0]}
  [462] = {x=10.077, y=0.000, z=-3.594, rx=-0.000, ry=0.000, rz=-0.000, shoulder=lefty, elbow=epositive, wrist=wnegative, fatherId=fReference[0]}
  [463] = {x=9.577, y=0.000, z=-3.601, rx=-0.000, ry=0.000, rz=-0.000, shoulder=lefty, elbow=epositive, wrist=wnegative, fatherId=fReference[0]}
  [464] = {x=9.077, y=0.000, z=-3.609, rx=-0.000, ry=0.000, rz=-0.000, shoulder=lefty, elbow=epositive, wrist=wnegative, fatherId=fReference[0]}
  [465] = {x=8.576, y=0.000, z=-3.617, rx=-0.000, ry=0.000, rz=-0.000, shoulder=lefty, elbow=epositive, wrist=wnegative, fatherId=fReference[0]}
  [466] = {x=8.076, y=0.000, z=-3.625, rx=-0.000, ry=0.000, rz=-0.000, shoulder=lefty, elbow=epositive, wrist=wnegative, fatherId=fReference[0]}
  [467] = {x=7.576, y=0.000, z=-3.633, rx=-0.000, ry=0.000, rz=-0.000, shoulder=lefty, elbow=epositive, wrist=wnegative, fatherId=fReference[0]}
  [468] = {x=7.076, y=0.000, z=-3.641, rx=-0.000, ry=0.000, rz=-0.000, shoulder=lefty, elbow=epositive, wrist=wnegative, fatherId=fReference[0]}
  [469] = {x=6.576, y=0.000, z=-3.649, rx=-0.000, ry=0.000, rz=-0.000, shoulder=lefty, elbow=epositive, wrist=wnegative, fatherId=fReference[0]}
  [470] = {x=6.076, y=0.000, z=-3.657, rx=-0.000, ry=0.000, rz=-0.000, shoulder=lefty, elbow=epositive, wrist=wnegative, fatherId=fReference[0]}
  [471] = {x=5.575, y=0.000, z=-3.666, rx=-0.000, ry=0.000, rz=-0.000, shoulder=lefty, elbow=epositive, wrist=wnegative, fatherId=fReference[0]}
  [472] = {x=5.075, y=0.000, z=-3.674, rx=-0.000, ry=0.000, rz=-0.000, shoulder=lefty, elbow=epositive, wrist=wnegative, fatherId=fReference[0]}
  [473] = {x=4.575, y=0.000, z=-3.682, rx=-0.000, ry=0.000, rz=-0.000, shoulder=lefty, elbow=epositive, wrist=wnegative, fatherId=fReference[0]}
  [474] = {x=4.075, y=0.000, z=-3.690, rx=-0.000, ry=0.000, rz=-0.000, shoulder=lefty, elbow=epositive, wrist=wnegative, fatherId=fReference[0]}
  [475] = {x=3.575, y=0.000, z=-3.698, rx=-0.000, ry=0.000, rz=-0.000, shoulder=lefty, elbow=epositive, wrist=wnegative, fatherId=fReference[0]}
  [476] = {x=3.074, y=0.000, z=-3.706, rx=-0.000, ry=0.000, rz=-0.000, shoulder=lefty, elbow=epositive, wrist=wnegative, fatherId=fReference[0]}
  [477] = {x=2.574, y=0.000, z=-3.715, rx=-0.000, ry=0.000, rz=-0.000, shoulder=lefty, elbow=epositive, wrist=wnegative, fatherId=fReference[0]}
  [478] = {x=2.074, y=0.000, z=-3.723, rx=-0.000, ry=0.000, rz=-0.000, shoulder=lefty, elbow=epositive, wrist=wnegative, fatherId=fReference[0]}
  [479] = {x=1.574, y=0.000, z=-3.732, rx=-0.000, ry=0.000, rz=-0.000, shoulder=lefty, elbow=epositive, wrist=wnegative, fatherId=fReference[0]}
  [480] = {x=1.074, y=0.000, z=-3.740, rx=-0.000, ry=0.000, rz=-0.000, shoulder=lefty, elbow=epositive, wrist=wnegative, fatherId=fReference[0]}
  [481] = {x=0.574, y=0.000, z=-3.748, rx=-0.000, ry=0.000, rz=-0.000, shoulder=lefty, elbow=epositive, wrist=wnegative, fatherId=fReference[0]}
  [482] = {x=0.074, y=0.000, z=-3.757, rx=-0.000, ry=0.000, rz=-0.000, shoulder=lefty, elbow=epositive, wrist=wnegative, fatherId=fReference[0]}
  [483] = {x=-0.426, y=0.000, z=-3.765, rx=-0.000, ry=0.000, rz=-0.000, shoulder=lefty, elbow=epositive, wrist=wnegative, fatherId=fReference[0]}
  [484] = {x=-0.926, y=0.000, z=-3.774, rx=-0.000, ry=0.000, rz=-0.000, shoulder=lefty, elbow=epositive, wrist=wnegative, fatherId=fReference[0]}
  [485] = {x=-1.426, y=0.000, z=-3.783, rx=-0.000, ry=0.000, rz=-0.000, shoulder=lefty, elbow=epositive, wrist=wnegative, fatherId=fReference[0]}
  [486] = {x=-1.926, y=0.000, z=-3.791, rx=-0.000, ry=0.000, rz=-0.000, shoulder=lefty, elbow=epositive, wrist=wnegative, fatherId=fReference[0]}
  [487] = {x=-2.426, y=0.000, z=-3.800, rx=-0.000, ry=0.000, rz=-0.000, shoulder=lefty, elbow=epositive, wrist=wnegative, fatherId=fReference[0]}
  [488] = {x=-2.926, y=0.000, z=-3.809, rx=-0.000, ry=0.000, rz=-0.000, shoulder=lefty, elbow=epositive, wrist=wnegative, fatherId=fReference[0]}
  [489] = {x=-3.426, y=0.000, z=-3.817, rx=-0.000, ry=0.000, rz=-0.000, shoulder=lefty, elbow=epositive, wrist=wnegative, fatherId=fReference[0]}
  [490] = {x=-3.927, y=0.000, z=-3.826, rx=-0.000, ry=0.000, rz=-0.000, shoulder=lefty, elbow=epositive, wrist=wnegative, fatherId=fReference[0]}
  [491] = {x=-4.427, y=0.000, z=-3.834, rx=-0.000, ry=0.000, rz=-0.000, shoulder=lefty, elbow=epositive, wrist=wnegative, fatherId=fReference[0]}
  [492] = {x=-4.927, y=0.000, z=-3.843, rx=-0.000, ry=0.000, rz=-0.000, shoulder=lefty, elbow=epositive, wrist=wnegative, fatherId=fReference[0]}
  [493] = {x=-5.427, y=0.000, z=-3.852, rx=-0.000, ry=0.000, rz=-0.000, shoulder=lefty, elbow=epositive, wrist=wnegative, fatherId=fReference[0]}
  [494] = {x=-5.927, y=0.000, z=-3.860, rx=-0.000, ry=0.000, rz=-0.000, shoulder=lefty, elbow=epositive, wrist=wnegative, fatherId=fReference[0]}
  [495] = {x=-6.427, y=0.000, z=-3.869, rx=-0.000, ry=0.000, rz=-0.000, shoulder=lefty, elbow=epositive, wrist=wnegative, fatherId=fReference[0]}
  [496] = {x=-6.927, y=0.000, z=-3.878, rx=-0.000, ry=0.000, rz=-0.000, shoulder=lefty, elbow=epositive, wrist=wnegative, fatherId=fReference[0]}
  [497] = {x=-7.428, y=0.000, z=-3.887, rx=-0.000, ry=0.000, rz=-0.000, shoulder=lefty, elbow=epositive, wrist=wnegative, fatherId=fReference[0]}
  [498] = {x=-7.928, y=0.000, z=-3.895, rx=-0.000, ry=0.000, rz=-0.000, shoulder=lefty, elbow=epositive, wrist=wnegative, fatherId=fReference[0]}
  [499] = {x=-8.428, y=0.000, z=-3.904, rx=-0.000, ry=0.000, rz=-0.000, shoulder=lefty, elbow=epositive, wrist=wnegative, fatherId=fReference[0]}
  [500] = {x=-8.929, y=0.000, z=-3.912, rx=-0.000, ry=0.000, rz=-0.000, shoulder=lefty, elbow=epositive, wrist=wnegative, fatherId=fReference[0]}
  [501] = {x=-9.429, y=0.000, z=-3.921, rx=-0.000, ry=0.000, rz=-0.000, shoulder=lefty, elbow=epositive, wrist=wnegative, fatherId=fReference[0]}
  [502] = {x=-9.930, y=0.000, z=-3.930, rx=-0.000, ry=0.000, rz=-0.000, shoulder=lefty, elbow=epositive, wrist=wnegative, fatherId=fReference[0]}
  [503] = {x=-10.430, y=0.000, z=-3.938, rx=-0.000, ry=0.000, rz=-0.000, shoulder=lefty, elbow=epositive, wrist=wnegative, fatherId=fReference[0]}
  [504] = {x=-10.930, y=0.000, z=-3.947, rx=-0.000, ry=0.000, rz=-0.000, shoulder=lefty, elbow=epositive, wrist=wnegative, fatherId=fReference[0]}
  [505] = {x=-11.431, y=0.000, z=-3.956, rx=-0.000, ry=0.000, rz=-0.000, shoulder=lefty, elbow=epositive, wrist=wnegative, fatherId=fReference[0]}
  [506] = {x=-11.931, y=0.000, z=-3.965, rx=-0.000, ry=0.000, rz=-0.000, shoulder=lefty, elbow=epositive, wrist=wnegative, fatherId=fReference[0]}
  [507] = {x=-12.431, y=0.000, z=-3.974, rx=-0.000, ry=0.000, rz=-0.000, shoulder=lefty, elbow=epositive, wrist=wnegative, fatherId=fReference[0]}
  [508] = {x=-12.932, y=0.000, z=-3.983, rx=-0.000, ry=0.000, rz=-0.000, shoulder=lefty, elbow=epositive, wrist=wnegative, fatherId=fReference[0]}
  [509] = {x=-13.432, y=0.000, z=-3.991, rx=-0.000, ry=0.000, rz=-0.000, shoulder=lefty, elbow=epositive, wrist=wnegative, fatherId=fReference[0]}
  [510] = {x=-13.932, y=0.000, z=-4.001, rx=-0.000, ry=0.000, rz=-0.000, shoulder=lefty, elbow=epositive, wrist=wnegative, fatherId=fReference[0]}
  [511] = {x=-14.432, y=0.000, z=-4.010, rx=-0.000, ry=0.000, rz=-0.000, shoulder=lefty, elbow=epositive, wrist=wnegative, fatherId=fReference[0]}
  [512] = {x=-14.933, y=0.000, z=-4.019, rx=-0.000, ry=0.000, rz=-0.000, shoulder=lefty, elbow=epositive, wrist=wnegative, fatherId=fReference[0]}
  [513] = {x=-15.433, y=0.000, z=-4.028, rx=-0.000, ry=0.000, rz=-0.000, shoulder=lefty, elbow=epositive, wrist=wnegative, fatherId=fReference[0]}
  [514] = {x=-15.934, y=0.000, z=-4.037, rx=-0.000, ry=0.000, rz=-0.000, shoulder=lefty, elbow=epositive, wrist=wnegative, fatherId=fReference[0]}
  [515] = {x=-16.434, y=0.000, z=-4.046, rx=-0.000, ry=0.000, rz=-0.000, shoulder=lefty, elbow=epositive, wrist=wnegative, fatherId=fReference[0]}
  [516] = {x=-16.935, y=0.000, z=-4.055, rx=-0.000, ry=0.000, rz=-0.000, shoulder=lefty, elbow=epositive, wrist=wnegative, fatherId=fReference[0]}
  [517] = {x=-17.435, y=0.000, z=-4.064, rx=-0.000, ry=0.000, rz=-0.000, shoulder=lefty, elbow=epositive, wrist=wnegative, fatherId=fReference[0]}
  [518] = {x=-17.936, y=0.000, z=-4.073, rx=-0.000, ry=0.000, rz=-0.000, shoulder=lefty, elbow=epositive, wrist=wnegative, fatherId=fReference[0]}
  [519] = {x=-18.436, y=0.000, z=-4.082, rx=-0.000, ry=0.000, rz=-0.000, shoulder=lefty, elbow=epositive, wrist=wnegative, fatherId=fReference[0]}
  [520] = {x=-18.937, y=0.000, z=-4.091, rx=-0.000, ry=0.000, rz=-0.000, shoulder=lefty, elbow=epositive, wrist=wnegative, fatherId=fReference[0]}
  [521] = {x=-19.437, y=0.000, z=-4.101, rx=-0.000, ry=0.000, rz=-0.000, shoulder=lefty, elbow=epositive, wrist=wnegative, fatherId=fReference[0]}
  [522] = {x=-19.938, y=0.000, z=-4.110, rx=-0.000, ry=0.000, rz=-0.000, shoulder=lefty, elbow=epositive, wrist=wnegative, fatherId=fReference[0]}
  [523] = {x=-20.438, y=0.000, z=-4.119, rx=-0.000, ry=0.000, rz=-0.000, shoulder=lefty, elbow=epositive, wrist=wnegative, fatherId=fReference[0]}
  [524] = {x=-20.938, y=0.000, z=-4.129, rx=-0.000, ry=0.000, rz=-0.000, shoulder=lefty, elbow=epositive, wrist=wnegative, fatherId=fReference[0]}
  [525] = {x=-21.439, y=0.000, z=-4.138, rx=-0.000, ry=0.000, rz=-0.000, shoulder=lefty, elbow=epositive, wrist=wnegative, fatherId=fReference[0]}
  [526] = {x=-21.940, y=0.000, z=-4.148, rx=-0.000, ry=0.000, rz=-0.000, shoulder=lefty, elbow=epositive, wrist=wnegative, fatherId=fReference[0]}
  [527] = {x=-22.441, y=0.000, z=-4.157, rx=-0.000, ry=0.000, rz=-0.000, shoulder=lefty, elbow=epositive, wrist=wnegative, fatherId=fReference[0]}
  [528] = {x=-22.940, y=0.000, z=-4.167, rx=-0.000, ry=0.000, rz=-0.000, shoulder=lefty, elbow=epositive, wrist=wnegative, fatherId=fReference[0]}
  [529] = {x=-23.442, y=0.000, z=-4.177, rx=-0.000, ry=0.000, rz=-0.000, shoulder=lefty, elbow=epositive, wrist=wnegative, fatherId=fReference[0]}
  [530] = {x=-23.943, y=0.000, z=-4.187, rx=-0.000, ry=0.000, rz=-0.000, shoulder=lefty, elbow=epositive, wrist=wnegative, fatherId=fReference[0]}
  [531] = {x=-24.442, y=0.000, z=-4.197, rx=-0.000, ry=0.000, rz=-0.000, shoulder=lefty, elbow=epositive, wrist=wnegative, fatherId=fReference[0]}
  [532] = {x=-24.943, y=0.000, z=-4.208, rx=-0.000, ry=0.000, rz=-0.000, shoulder=lefty, elbow=epositive, wrist=wnegative, fatherId=fReference[0]}
  [533] = {x=-25.443, y=0.000, z=-4.219, rx=-0.000, ry=0.000, rz=-0.000, shoulder=lefty, elbow=epositive, wrist=wnegative, fatherId=fReference[0]}
  [534] = {x=-25.944, y=0.000, z=-4.229, rx=-0.000, ry=0.000, rz=-0.000, shoulder=lefty, elbow=epositive, wrist=wnegative, fatherId=fReference[0]}
  [535] = {x=-26.443, y=0.000, z=-4.240, rx=-0.000, ry=0.000, rz=-0.000, shoulder=lefty, elbow=epositive, wrist=wnegative, fatherId=fReference[0]}
  [536] = {x=-26.943, y=0.000, z=-4.251, rx=-0.000, ry=0.000, rz=-0.000, shoulder=lefty, elbow=epositive, wrist=wnegative, fatherId=fReference[0]}
  [537] = {x=-27.444, y=0.000, z=-4.262, rx=-0.000, ry=0.000, rz=-0.000, shoulder=lefty, elbow=epositive, wrist=wnegative, fatherId=fReference[0]}
  [538] = {x=-27.944, y=0.000, z=-4.272, rx=-0.000, ry=0.000, rz=-0.000, shoulder=lefty, elbow=epositive, wrist=wnegative, fatherId=fReference[0]}
  [539] = {x=-28.444, y=0.000, z=-4.283, rx=-0.000, ry=0.000, rz=-0.000, shoulder=lefty, elbow=epositive, wrist=wnegative, fatherId=fReference[0]}
  [540] = {x=-28.944, y=0.000, z=-4.294, rx=-0.000, ry=0.000, rz=-0.000, shoulder=lefty, elbow=epositive, wrist=wnegative, fatherId=fReference[0]}
  [541] = {x=-29.445, y=0.000, z=-4.305, rx=-0.000, ry=0.000, rz=-0.000, shoulder=lefty, elbow=epositive, wrist=wnegative, fatherId=fReference[0]}
  [542] = {x=-29.945, y=0.000, z=-4.316, rx=-0.000, ry=0.000, rz=-0.000, shoulder=lefty, elbow=epositive, wrist=wnegative, fatherId=fReference[0]}
  [543] = {x=-30.445, y=0.000, z=-4.327, rx=-0.000, ry=0.000, rz=-0.000, shoulder=lefty, elbow=epositive, wrist=wnegative, fatherId=fReference[0]}
  [544] = {x=-30.946, y=0.000, z=-4.337, rx=-0.000, ry=0.000, rz=-0.000, shoulder=lefty, elbow=epositive, wrist=wnegative, fatherId=fReference[0]}
  [545] = {x=-31.448, y=0.000, z=-4.347, rx=-0.000, ry=0.000, rz=-0.000, shoulder=lefty, elbow=epositive, wrist=wnegative, fatherId=fReference[0]}
  [546] = {x=-31.951, y=0.000, z=-4.357, rx=-0.000, ry=0.000, rz=-0.000, shoulder=lefty, elbow=epositive, wrist=wnegative, fatherId=fReference[0]}
  [547] = {x=-32.455, y=0.000, z=-4.366, rx=-0.000, ry=0.000, rz=-0.000, shoulder=lefty, elbow=epositive, wrist=wnegative, fatherId=fReference[0]}
  [548] = {x=-32.834, y=0.000, z=-4.349, rx=-0.000, ry=0.000, rz=-0.000, shoulder=lefty, elbow=epositive, wrist=wnegative, fatherId=fReference[0]}
  [549] = {x=-32.323, y=0.000, z=-4.341, rx=-0.000, ry=0.000, rz=-0.000, shoulder=lefty, elbow=epositive, wrist=wnegative, fatherId=fReference[0]}
  [550] = {x=-31.819, y=0.000, z=-4.339, rx=-0.000, ry=0.000, rz=-0.000, shoulder=lefty, elbow=epositive, wrist=wnegative, fatherId=fReference[0]}
  [551] = {x=-31.316, y=0.000, z=-4.339, rx=-0.000, ry=0.000, rz=-0.000, shoulder=lefty, elbow=epositive, wrist=wnegative, fatherId=fReference[0]}
  [552] = {x=-30.814, y=0.000, z=-4.342, rx=-0.000, ry=0.000, rz=-0.000, shoulder=lefty, elbow=epositive, wrist=wnegative, fatherId=fReference[0]}
  [553] = {x=-30.313, y=0.000, z=-4.348, rx=-0.000, ry=0.000, rz=-0.000, shoulder=lefty, elbow=epositive, wrist=wnegative, fatherId=fReference[0]}
  [554] = {x=-29.811, y=0.000, z=-4.353, rx=-0.000, ry=0.000, rz=-0.000, shoulder=lefty, elbow=epositive, wrist=wnegative, fatherId=fReference[0]}
  [555] = {x=-29.310, y=0.000, z=-4.360, rx=-0.000, ry=0.000, rz=-0.000, shoulder=lefty, elbow=epositive, wrist=wnegative, fatherId=fReference[0]}
  [556] = {x=-28.809, y=0.000, z=-4.367, rx=-0.000, ry=0.000, rz=-0.000, shoulder=lefty, elbow=epositive, wrist=wnegative, fatherId=fReference[0]}
  [557] = {x=-28.308, y=0.000, z=-4.374, rx=-0.000, ry=0.000, rz=-0.000, shoulder=lefty, elbow=epositive, wrist=wnegative, fatherId=fReference[0]}
  [558] = {x=-27.807, y=0.000, z=-4.382, rx=-0.000, ry=0.000, rz=-0.000, shoulder=lefty, elbow=epositive, wrist=wnegative, fatherId=fReference[0]}
  [559] = {x=-27.306, y=0.000, z=-4.389, rx=-0.000, ry=0.000, rz=-0.000, shoulder=lefty, elbow=epositive, wrist=wnegative, fatherId=fReference[0]}
  [560] = {x=-26.805, y=0.000, z=-4.398, rx=-0.000, ry=0.000, rz=-0.000, shoulder=lefty, elbow=epositive, wrist=wnegative, fatherId=fReference[0]}
  [561] = {x=-26.305, y=0.000, z=-4.405, rx=-0.000, ry=0.000, rz=-0.000, shoulder=lefty, elbow=epositive, wrist=wnegative, fatherId=fReference[0]}
  [562] = {x=-25.803, y=0.000, z=-4.414, rx=-0.000, ry=0.000, rz=-0.000, shoulder=lefty, elbow=epositive, wrist=wnegative, fatherId=fReference[0]}
  [563] = {x=-25.302, y=0.000, z=-4.422, rx=-0.000, ry=0.000, rz=-0.000, shoulder=lefty, elbow=epositive, wrist=wnegative, fatherId=fReference[0]}
  [564] = {x=-24.801, y=0.000, z=-4.431, rx=-0.000, ry=0.000, rz=-0.000, shoulder=lefty, elbow=epositive, wrist=wnegative, fatherId=fReference[0]}
  [565] = {x=-24.300, y=0.000, z=-4.440, rx=-0.000, ry=0.000, rz=-0.000, shoulder=lefty, elbow=epositive, wrist=wnegative, fatherId=fReference[0]}
  [566] = {x=-23.799, y=0.000, z=-4.449, rx=-0.000, ry=0.000, rz=-0.000, shoulder=lefty, elbow=epositive, wrist=wnegative, fatherId=fReference[0]}
  [567] = {x=-23.297, y=0.000, z=-4.457, rx=-0.000, ry=0.000, rz=-0.000, shoulder=lefty, elbow=epositive, wrist=wnegative, fatherId=fReference[0]}
  [568] = {x=-22.795, y=0.000, z=-4.467, rx=-0.000, ry=0.000, rz=-0.000, shoulder=lefty, elbow=epositive, wrist=wnegative, fatherId=fReference[0]}
  [569] = {x=-22.294, y=0.000, z=-4.476, rx=-0.000, ry=0.000, rz=-0.000, shoulder=lefty, elbow=epositive, wrist=wnegative, fatherId=fReference[0]}
  [570] = {x=-21.793, y=0.000, z=-4.485, rx=-0.000, ry=0.000, rz=-0.000, shoulder=lefty, elbow=epositive, wrist=wnegative, fatherId=fReference[0]}
  [571] = {x=-21.292, y=0.000, z=-4.494, rx=-0.000, ry=0.000, rz=-0.000, shoulder=lefty, elbow=epositive, wrist=wnegative, fatherId=fReference[0]}
  [572] = {x=-20.791, y=0.000, z=-4.503, rx=-0.000, ry=0.000, rz=-0.000, shoulder=lefty, elbow=epositive, wrist=wnegative, fatherId=fReference[0]}
  [573] = {x=-20.289, y=0.000, z=-4.512, rx=-0.000, ry=0.000, rz=-0.000, shoulder=lefty, elbow=epositive, wrist=wnegative, fatherId=fReference[0]}
  [574] = {x=-19.788, y=0.000, z=-4.521, rx=-0.000, ry=0.000, rz=-0.000, shoulder=lefty, elbow=epositive, wrist=wnegative, fatherId=fReference[0]}
  [575] = {x=-19.287, y=0.000, z=-4.529, rx=-0.000, ry=0.000, rz=-0.000, shoulder=lefty, elbow=epositive, wrist=wnegative, fatherId=fReference[0]}
  [576] = {x=-18.785, y=0.000, z=-4.538, rx=-0.000, ry=0.000, rz=-0.000, shoulder=lefty, elbow=epositive, wrist=wnegative, fatherId=fReference[0]}
  [577] = {x=-18.284, y=0.000, z=-4.547, rx=-0.000, ry=0.000, rz=-0.000, shoulder=lefty, elbow=epositive, wrist=wnegative, fatherId=fReference[0]}
  [578] = {x=-17.783, y=0.000, z=-4.556, rx=-0.000, ry=0.000, rz=-0.000, shoulder=lefty, elbow=epositive, wrist=wnegative, fatherId=fReference[0]}
  [579] = {x=-17.281, y=0.000, z=-4.564, rx=-0.000, ry=0.000, rz=-0.000, shoulder=lefty, elbow=epositive, wrist=wnegative, fatherId=fReference[0]}
  [580] = {x=-16.779, y=0.000, z=-4.573, rx=-0.000, ry=0.000, rz=-0.000, shoulder=lefty, elbow=epositive, wrist=wnegative, fatherId=fReference[0]}
  [581] = {x=-16.278, y=0.000, z=-4.582, rx=-0.000, ry=0.000, rz=-0.000, shoulder=lefty, elbow=epositive, wrist=wnegative, fatherId=fReference[0]}
  [582] = {x=-15.777, y=0.000, z=-4.590, rx=-0.000, ry=0.000, rz=-0.000, shoulder=lefty, elbow=epositive, wrist=wnegative, fatherId=fReference[0]}
  [583] = {x=-15.276, y=0.000, z=-4.599, rx=-0.000, ry=0.000, rz=-0.000, shoulder=lefty, elbow=epositive, wrist=wnegative, fatherId=fReference[0]}
  [584] = {x=-14.775, y=0.000, z=-4.607, rx=-0.000, ry=0.000, rz=-0.000, shoulder=lefty, elbow=epositive, wrist=wnegative, fatherId=fReference[0]}
  [585] = {x=-14.273, y=0.000, z=-4.615, rx=-0.000, ry=0.000, rz=-0.000, shoulder=lefty, elbow=epositive, wrist=wnegative, fatherId=fReference[0]}
  [586] = {x=-13.773, y=0.000, z=-4.624, rx=-0.000, ry=0.000, rz=-0.000, shoulder=lefty, elbow=epositive, wrist=wnegative, fatherId=fReference[0]}
  [587] = {x=-13.272, y=0.000, z=-4.632, rx=-0.000, ry=0.000, rz=-0.000, shoulder=lefty, elbow=epositive, wrist=wnegative, fatherId=fReference[0]}
  [588] = {x=-12.770, y=0.000, z=-4.640, rx=-0.000, ry=0.000, rz=-0.000, shoulder=lefty, elbow=epositive, wrist=wnegative, fatherId=fReference[0]}
  [589] = {x=-12.269, y=0.000, z=-4.648, rx=-0.000, ry=0.000, rz=-0.000, shoulder=lefty, elbow=epositive, wrist=wnegative, fatherId=fReference[0]}
  [590] = {x=-11.768, y=0.000, z=-4.656, rx=-0.000, ry=0.000, rz=-0.000, shoulder=lefty, elbow=epositive, wrist=wnegative, fatherId=fReference[0]}
  [591] = {x=-11.267, y=0.000, z=-4.665, rx=-0.000, ry=0.000, rz=-0.000, shoulder=lefty, elbow=epositive, wrist=wnegative, fatherId=fReference[0]}
  [592] = {x=-10.766, y=0.000, z=-4.673, rx=-0.000, ry=0.000, rz=-0.000, shoulder=lefty, elbow=epositive, wrist=wnegative, fatherId=fReference[0]}
  [593] = {x=-10.264, y=0.000, z=-4.681, rx=-0.000, ry=0.000, rz=-0.000, shoulder=lefty, elbow=epositive, wrist=wnegative, fatherId=fReference[0]}
  [594] = {x=-9.763, y=0.000, z=-4.689, rx=-0.000, ry=0.000, rz=-0.000, shoulder=lefty, elbow=epositive, wrist=wnegative, fatherId=fReference[0]}
  [595] = {x=-9.262, y=0.000, z=-4.697, rx=-0.000, ry=0.000, rz=-0.000, shoulder=lefty, elbow=epositive, wrist=wnegative, fatherId=fReference[0]}
  [596] = {x=-8.761, y=0.000, z=-4.705, rx=-0.000, ry=0.000, rz=-0.000, shoulder=lefty, elbow=epositive, wrist=wnegative, fatherId=fReference[0]}
  [597] = {x=-8.260, y=0.000, z=-4.713, rx=-0.000, ry=0.000, rz=-0.000, shoulder=lefty, elbow=epositive, wrist=wnegative, fatherId=fReference[0]}
  [598] = {x=-7.759, y=0.000, z=-4.721, rx=-0.000, ry=0.000, rz=-0.000, shoulder=lefty, elbow=epositive, wrist=wnegative, fatherId=fReference[0]}
  [599] = {x=-7.258, y=0.000, z=-4.729, rx=-0.000, ry=0.000, rz=-0.000, shoulder=lefty, elbow=epositive, wrist=wnegative, fatherId=fReference[0]}
  [600] = {x=-6.757, y=0.000, z=-4.737, rx=-0.000, ry=0.000, rz=-0.000, shoulder=lefty, elbow=epositive, wrist=wnegative, fatherId=fReference[0]}
  [601] = {x=-6.256, y=0.000, z=-4.745, rx=-0.000, ry=0.000, rz=-0.000, shoulder=lefty, elbow=epositive, wrist=wnegative, fatherId=fReference[0]}
  [602] = {x=-5.755, y=0.000, z=-4.753, rx=-0.000, ry=0.000, rz=-0.000, shoulder=lefty, elbow=epositive, wrist=wnegative, fatherId=fReference[0]}
  [603] = {x=-5.254, y=0.000, z=-4.760, rx=-0.000, ry=0.000, rz=-0.000, shoulder=lefty, elbow=epositive, wrist=wnegative, fatherId=fReference[0]}
  [604] = {x=-4.753, y=0.000, z=-4.768, rx=-0.000, ry=0.000, rz=-0.000, shoulder=lefty, elbow=epositive, wrist=wnegative, fatherId=fReference[0]}
  [605] = {x=-4.252, y=0.000, z=-4.776, rx=-0.000, ry=0.000, rz=-0.000, shoulder=lefty, elbow=epositive, wrist=wnegative, fatherId=fReference[0]}
  [606] = {x=-3.751, y=0.000, z=-4.784, rx=-0.000, ry=0.000, rz=-0.000, shoulder=lefty, elbow=epositive, wrist=wnegative, fatherId=fReference[0]}
  [607] = {x=-3.250, y=0.000, z=-4.792, rx=-0.000, ry=0.000, rz=-0.000, shoulder=lefty, elbow=epositive, wrist=wnegative, fatherId=fReference[0]}
  [608] = {x=-2.749, y=0.000, z=-4.800, rx=-0.000, ry=0.000, rz=-0.000, shoulder=lefty, elbow=epositive, wrist=wnegative, fatherId=fReference[0]}
  [609] = {x=-2.248, y=0.000, z=-4.808, rx=-0.000, ry=0.000, rz=-0.000, shoulder=lefty, elbow=epositive, wrist=wnegative, fatherId=fReference[0]}
  [610] = {x=-1.747, y=0.000, z=-4.816, rx=-0.000, ry=0.000, rz=-0.000, shoulder=lefty, elbow=epositive, wrist=wnegative, fatherId=fReference[0]}
  [611] = {x=-1.245, y=0.000, z=-4.824, rx=-0.000, ry=0.000, rz=-0.000, shoulder=lefty, elbow=epositive, wrist=wnegative, fatherId=fReference[0]}
  [612] = {x=-0.744, y=0.000, z=-4.832, rx=-0.000, ry=0.000, rz=-0.000, shoulder=lefty, elbow=epositive, wrist=wnegative, fatherId=fReference[0]}
  [613] = {x=-0.243, y=0.000, z=-4.841, rx=-0.000, ry=0.000, rz=-0.000, shoulder=lefty, elbow=epositive, wrist=wnegative, fatherId=fReference[0]}
  [614] = {x=0.259, y=0.000, z=-4.849, rx=-0.000, ry=0.000, rz=-0.000, shoulder=lefty, elbow=epositive, wrist=wnegative, fatherId=fReference[0]}
  [615] = {x=0.760, y=0.000, z=-4.858, rx=-0.000, ry=0.000, rz=-0.000, shoulder=lefty, elbow=epositive, wrist=wnegative, fatherId=fReference[0]}
  [616] = {x=1.262, y=0.000, z=-4.866, rx=-0.000, ry=0.000, rz=-0.000, shoulder=lefty, elbow=epositive, wrist=wnegative, fatherId=fReference[0]}
  [617] = {x=1.764, y=0.000, z=-4.874, rx=-0.000, ry=0.000, rz=-0.000, shoulder=lefty, elbow=epositive, wrist=wnegative, fatherId=fReference[0]}
  [618] = {x=2.266, y=0.000, z=-4.882, rx=-0.000, ry=0.000, rz=-0.000, shoulder=lefty, elbow=epositive, wrist=wnegative, fatherId=fReference[0]}
  [619] = {x=2.767, y=0.000, z=-4.890, rx=-0.000, ry=0.000, rz=-0.000, shoulder=lefty, elbow=epositive, wrist=wnegative, fatherId=fReference[0]}
  [620] = {x=3.269, y=0.000, z=-4.898, rx=-0.000, ry=0.000, rz=-0.000, shoulder=lefty, elbow=epositive, wrist=wnegative, fatherId=fReference[0]}
  [621] = {x=3.771, y=0.000, z=-4.907, rx=-0.000, ry=0.000, rz=-0.000, shoulder=lefty, elbow=epositive, wrist=wnegative, fatherId=fReference[0]}
  [622] = {x=4.272, y=0.000, z=-4.915, rx=-0.000, ry=0.000, rz=-0.000, shoulder=lefty, elbow=epositive, wrist=wnegative, fatherId=fReference[0]}
  [623] = {x=4.774, y=0.000, z=-4.924, rx=-0.000, ry=0.000, rz=-0.000, shoulder=lefty, elbow=epositive, wrist=wnegative, fatherId=fReference[0]}
  [624] = {x=5.276, y=0.000, z=-4.932, rx=-0.000, ry=0.000, rz=-0.000, shoulder=lefty, elbow=epositive, wrist=wnegative, fatherId=fReference[0]}
  [625] = {x=5.778, y=0.000, z=-4.941, rx=-0.000, ry=0.000, rz=-0.000, shoulder=lefty, elbow=epositive, wrist=wnegative, fatherId=fReference[0]}
  [626] = {x=6.279, y=0.000, z=-4.949, rx=-0.000, ry=0.000, rz=-0.000, shoulder=lefty, elbow=epositive, wrist=wnegative, fatherId=fReference[0]}
  [627] = {x=6.781, y=0.000, z=-4.958, rx=-0.000, ry=0.000, rz=-0.000, shoulder=lefty, elbow=epositive, wrist=wnegative, fatherId=fReference[0]}
  [628] = {x=7.283, y=0.000, z=-4.967, rx=-0.000, ry=0.000, rz=-0.000, shoulder=lefty, elbow=epositive, wrist=wnegative, fatherId=fReference[0]}
  [629] = {x=7.785, y=0.000, z=-4.976, rx=-0.000, ry=0.000, rz=-0.000, shoulder=lefty, elbow=epositive, wrist=wnegative, fatherId=fReference[0]}
  [630] = {x=8.287, y=0.000, z=-4.985, rx=-0.000, ry=0.000, rz=-0.000, shoulder=lefty, elbow=epositive, wrist=wnegative, fatherId=fReference[0]}
  [631] = {x=8.789, y=0.000, z=-4.994, rx=-0.000, ry=0.000, rz=-0.000, shoulder=lefty, elbow=epositive, wrist=wnegative, fatherId=fReference[0]}
  [632] = {x=9.291, y=0.000, z=-5.003, rx=-0.000, ry=0.000, rz=-0.000, shoulder=lefty, elbow=epositive, wrist=wnegative, fatherId=fReference[0]}
  [633] = {x=9.793, y=0.000, z=-5.012, rx=-0.000, ry=0.000, rz=-0.000, shoulder=lefty, elbow=epositive, wrist=wnegative, fatherId=fReference[0]}
  [634] = {x=10.296, y=0.000, z=-5.021, rx=-0.000, ry=0.000, rz=-0.000, shoulder=lefty, elbow=epositive, wrist=wnegative, fatherId=fReference[0]}
  [635] = {x=10.798, y=0.000, z=-5.030, rx=-0.000, ry=0.000, rz=-0.000, shoulder=lefty, elbow=epositive, wrist=wnegative, fatherId=fReference[0]}
  [636] = {x=11.300, y=0.000, z=-5.040, rx=-0.000, ry=0.000, rz=-0.000, shoulder=lefty, elbow=epositive, wrist=wnegative, fatherId=fReference[0]}
  [637] = {x=11.803, y=0.000, z=-5.049, rx=-0.000, ry=0.000, rz=-0.000, shoulder=lefty, elbow=epositive, wrist=wnegative, fatherId=fReference[0]}
  [638] = {x=12.306, y=0.000, z=-5.058, rx=-0.000, ry=0.000, rz=-0.000, shoulder=lefty, elbow=epositive, wrist=wnegative, fatherId=fReference[0]}
  [639] = {x=12.808, y=0.000, z=-5.068, rx=-0.000, ry=0.000, rz=-0.000, shoulder=lefty, elbow=epositive, wrist=wnegative, fatherId=fReference[0]}
  [640] = {x=13.310, y=0.000, z=-5.077, rx=-0.000, ry=0.000, rz=-0.000, shoulder=lefty, elbow=epositive, wrist=wnegative, fatherId=fReference[0]}
  [641] = {x=13.813, y=0.000, z=-5.087, rx=-0.000, ry=0.000, rz=-0.000, shoulder=lefty, elbow=epositive, wrist=wnegative, fatherId=fReference[0]}
  [642] = {x=14.315, y=0.000, z=-5.097, rx=-0.000, ry=0.000, rz=-0.000, shoulder=lefty, elbow=epositive, wrist=wnegative, fatherId=fReference[0]}
  [643] = {x=14.818, y=0.000, z=-5.106, rx=-0.000, ry=0.000, rz=-0.000, shoulder=lefty, elbow=epositive, wrist=wnegative, fatherId=fReference[0]}
  [644] = {x=15.320, y=0.000, z=-5.116, rx=-0.000, ry=0.000, rz=-0.000, shoulder=lefty, elbow=epositive, wrist=wnegative, fatherId=fReference[0]}
  [645] = {x=15.823, y=0.000, z=-5.126, rx=-0.000, ry=0.000, rz=-0.000, shoulder=lefty, elbow=epositive, wrist=wnegative, fatherId=fReference[0]}
  [646] = {x=16.325, y=0.000, z=-5.135, rx=-0.000, ry=0.000, rz=-0.000, shoulder=lefty, elbow=epositive, wrist=wnegative, fatherId=fReference[0]}
  [647] = {x=16.829, y=0.000, z=-5.145, rx=-0.000, ry=0.000, rz=-0.000, shoulder=lefty, elbow=epositive, wrist=wnegative, fatherId=fReference[0]}
  [648] = {x=17.331, y=0.000, z=-5.155, rx=-0.000, ry=0.000, rz=-0.000, shoulder=lefty, elbow=epositive, wrist=wnegative, fatherId=fReference[0]}
  [649] = {x=17.833, y=0.000, z=-5.165, rx=-0.000, ry=0.000, rz=-0.000, shoulder=lefty, elbow=epositive, wrist=wnegative, fatherId=fReference[0]}
  [650] = {x=18.336, y=0.000, z=-5.175, rx=-0.000, ry=0.000, rz=-0.000, shoulder=lefty, elbow=epositive, wrist=wnegative, fatherId=fReference[0]}
  [651] = {x=18.839, y=0.000, z=-5.186, rx=-0.000, ry=0.000, rz=-0.000, shoulder=lefty, elbow=epositive, wrist=wnegative, fatherId=fReference[0]}
  [652] = {x=19.342, y=0.000, z=-5.196, rx=-0.000, ry=0.000, rz=-0.000, shoulder=lefty, elbow=epositive, wrist=wnegative, fatherId=fReference[0]}
  [653] = {x=19.845, y=0.000, z=-5.207, rx=-0.000, ry=0.000, rz=-0.000, shoulder=lefty, elbow=epositive, wrist=wnegative, fatherId=fReference[0]}
  [654] = {x=20.348, y=0.000, z=-5.218, rx=-0.000, ry=0.000, rz=-0.000, shoulder=lefty, elbow=epositive, wrist=wnegative, fatherId=fReference[0]}
  [655] = {x=20.851, y=0.000, z=-5.229, rx=-0.000, ry=0.000, rz=-0.000, shoulder=lefty, elbow=epositive, wrist=wnegative, fatherId=fReference[0]}
  [656] = {x=21.354, y=0.000, z=-5.239, rx=-0.000, ry=0.000, rz=-0.000, shoulder=lefty, elbow=epositive, wrist=wnegative, fatherId=fReference[0]}
  [657] = {x=21.856, y=0.000, z=-5.250, rx=-0.000, ry=0.000, rz=-0.000, shoulder=lefty, elbow=epositive, wrist=wnegative, fatherId=fReference[0]}
  [658] = {x=22.359, y=0.000, z=-5.261, rx=-0.000, ry=0.000, rz=-0.000, shoulder=lefty, elbow=epositive, wrist=wnegative, fatherId=fReference[0]}
  [659] = {x=22.863, y=0.000, z=-5.272, rx=-0.000, ry=0.000, rz=-0.000, shoulder=lefty, elbow=epositive, wrist=wnegative, fatherId=fReference[0]}
  [660] = {x=23.366, y=0.000, z=-5.283, rx=-0.000, ry=0.000, rz=-0.000, shoulder=lefty, elbow=epositive, wrist=wnegative, fatherId=fReference[0]}
  [661] = {x=23.869, y=0.000, z=-5.295, rx=-0.000, ry=0.000, rz=-0.000, shoulder=lefty, elbow=epositive, wrist=wnegative, fatherId=fReference[0]}
  [662] = {x=24.373, y=0.000, z=-5.306, rx=-0.000, ry=0.000, rz=-0.000, shoulder=lefty, elbow=epositive, wrist=wnegative, fatherId=fReference[0]}
  [663] = {x=24.876, y=0.000, z=-5.317, rx=-0.000, ry=0.000, rz=-0.000, shoulder=lefty, elbow=epositive, wrist=wnegative, fatherId=fReference[0]}
  [664] = {x=25.380, y=0.000, z=-5.328, rx=-0.000, ry=0.000, rz=-0.000, shoulder=lefty, elbow=epositive, wrist=wnegative, fatherId=fReference[0]}
  [665] = {x=25.884, y=0.000, z=-5.340, rx=-0.000, ry=0.000, rz=-0.000, shoulder=lefty, elbow=epositive, wrist=wnegative, fatherId=fReference[0]}
  [666] = {x=26.388, y=0.000, z=-5.351, rx=-0.000, ry=0.000, rz=-0.000, shoulder=lefty, elbow=epositive, wrist=wnegative, fatherId=fReference[0]}
  [667] = {x=26.892, y=0.000, z=-5.362, rx=-0.000, ry=0.000, rz=-0.000, shoulder=lefty, elbow=epositive, wrist=wnegative, fatherId=fReference[0]}
  [668] = {x=27.397, y=0.000, z=-5.374, rx=-0.000, ry=0.000, rz=-0.000, shoulder=lefty, elbow=epositive, wrist=wnegative, fatherId=fReference[0]}
  [669] = {x=27.902, y=0.000, z=-5.385, rx=-0.000, ry=0.000, rz=-0.000, shoulder=lefty, elbow=epositive, wrist=wnegative, fatherId=fReference[0]}
  [670] = {x=28.406, y=0.000, z=-5.397, rx=-0.000, ry=0.000, rz=-0.000, shoulder=lefty, elbow=epositive, wrist=wnegative, fatherId=fReference[0]}
  [671] = {x=28.911, y=0.000, z=-5.408, rx=-0.000, ry=0.000, rz=-0.000, shoulder=lefty, elbow=epositive, wrist=wnegative, fatherId=fReference[0]}
  [672] = {x=29.416, y=0.000, z=-5.419, rx=-0.000, ry=0.000, rz=-0.000, shoulder=lefty, elbow=epositive, wrist=wnegative, fatherId=fReference[0]}
  [673] = {x=29.922, y=0.000, z=-5.430, rx=-0.000, ry=0.000, rz=-0.000, shoulder=lefty, elbow=epositive, wrist=wnegative, fatherId=fReference[0]}
  [674] = {x=30.430, y=0.000, z=-5.441, rx=-0.000, ry=0.000, rz=-0.000, shoulder=lefty, elbow=epositive, wrist=wnegative, fatherId=fReference[0]}
  [675] = {x=30.936, y=0.000, z=-5.451, rx=-0.000, ry=0.000, rz=-0.000, shoulder=lefty, elbow=epositive, wrist=wnegative, fatherId=fReference[0]}
  [676] = {x=31.443, y=0.000, z=-5.459, rx=-0.000, ry=0.000, rz=-0.000, shoulder=lefty, elbow=epositive, wrist=wnegative, fatherId=fReference[0]}
  [677] = {x=31.949, y=0.000, z=-5.466, rx=-0.000, ry=0.000, rz=-0.000, shoulder=lefty, elbow=epositive, wrist=wnegative, fatherId=fReference[0]}
  [678] = {x=32.458, y=0.000, z=-5.472, rx=-0.000, ry=0.000, rz=-0.000, shoulder=lefty, elbow=epositive, wrist=wnegative, fatherId=fReference[0]}
  [679] = {x=32.967, y=0.000, z=-5.478, rx=-0.000, ry=0.000, rz=-0.000, shoulder=lefty, elbow=epositive, wrist=wnegative, fatherId=fReference[0]}
